gfCNCPoint3[12067] = {X 589.3965, Y 44.0652, Z -3.8333, A 0.000, B 0.000, C 0.000 }
gfCNCPoint3[12068] = {X 589.5012, Y 43.1533, Z -3.8333, A 0.000, B 0.000, C 0.000 }
gfCNCPoint3[12069] = {X 589.8014, Y 42.2858, Z -3.8333, A 0.000, B 0.000, C 0.000 }
gfCNCPoint3[12070] = {X 590.2828, Y 41.5042, Z -3.8333, A 0.000, B 0.000, C 0.000 }
gfCNCPoint3[12071] = {X 590.9225, Y 40.8459, Z -3.8333, A 0.000, B 0.000, C 0.000 }
gfCNCPoint3[12072] = {X 590.9230, Y 32.7095, Z -3.8333, A 0.000, B 0.000, C 0.000 }
gfCNCPoint3[12073] = {X 585.2975, Y 46.5912, Z -3.8333, A 0.000, B 0.000, C 0.000 }
gfCNCPoint3[12074] = {X 584.9414, Y 47.2678, Z -3.8333, A 0.000, B 0.000, C 0.000 }
gfCNCPoint3[12075] = {X 584.4675, Y 47.8677, Z -3.8333, A 0.000, B 0.000, C 0.000 }
gfCNCPoint3[12076] = {X 583.8918, Y 48.3708, Z -3.8333, A 0.000, B 0.000, C 0.000 }
gfCNCPoint3[12077] = {X 583.2338, Y 48.7600, Z -3.8333, A 0.000, B 0.000, C 0.000 }
gfCNCPoint3[12078] = {X 582.3250, Y 49.0678, Z -3.8333, A 0.000, B 0.000, C 0.000 }
gfCNCPoint3[12079] = {X 581.3699, Y 49.1592, Z -3.8333, A 0.000, B 0.000, C 0.000 }
gfCNCPoint3[12080] = {X 580.4192, Y 49.0293, Z -3.8333, A 0.000, B 0.000, C 0.000 }
gfCNCPoint3[12081] = {X 579.5236, Y 48.6850, Z -3.8333, A 0.000, B 0.000, C 0.000 }
gfCNCPoint3[12082] = {X 578.7306, Y 48.1448, Z -3.8333, A 0.000, B 0.000, C 0.000 }
gfCNCPoint3[12083] = {X 578.0826, Y 47.4372, Z -3.8333, A 0.000, B 0.000, C 0.000 }
gfCNCPoint3[12084] = {X 577.6138, Y 46.5999, Z -3.8333, A 0.000, B 0.000, C 0.000 }
gfCNCPoint3[12085] = {X 571.8585, Y 32.5267, Z -3.8333, A 0.000, B 0.000, C 0.000 }
gfCNCPoint3[12086] = {X 571.8589, Y 40.8461, Z -3.8333, A 0.000, B 0.000, C 0.000 }
gfCNCPoint3[12087] = {X 571.9195, Y 40.8953, Z -3.8333, A 0.000, B 0.000, C 0.000 }
gfCNCPoint3[12088] = {X 572.5327, Y 41.5413, Z -3.8333, A 0.000, B 0.000, C 0.000 }
gfCNCPoint3[12089] = {X 572.9944, Y 42.3029, Z -3.8333, A 0.000, B 0.000, C 0.000 }
gfCNCPoint3[12090] = {X 573.2833, Y 43.1454, Z -3.8333, A 0.000, B 0.000, C 0.000 }
gfCNCPoint3[12091] = {X 573.3863, Y 44.0301, Z -3.8333, A 0.000, B 0.000, C 0.000 }
gfCNCPoint3[12092] = {X 573.3864, Y 45.0000, Z -3.8333, A 0.000, B 0.000, C 0.000 }
gfCNCPoint3[12093] = {X 573.2821, Y 45.9257, Z -3.8333, A 0.000, B 0.000, C 0.000 }
gfCNCPoint3[12094] = {X 572.9745, Y 46.8050, Z -3.8333, A 0.000, B 0.000, C 0.000 }
gfCNCPoint3[12095] = {X 572.4788, Y 47.5937, Z -3.8333, A 0.000, B 0.000, C 0.000 }
gfCNCPoint3[12096] = {X 571.8201, Y 48.2524, Z -3.8333, A 0.000, B 0.000, C 0.000 }
gfCNCPoint3[12097] = {X 571.0314, Y 48.7480, Z -3.8333, A 0.000, B 0.000, C 0.000 }
gfCNCPoint3[12098] = {X 570.1521, Y 49.0557, Z -3.8333, A 0.000, B 0.000, C 0.000 }
gfCNCPoint3[12099] = {X 569.2264, Y 49.1600, Z -3.8333, A 0.000, B 0.000, C 0.000 }
gfCNCPoint3[12100] = {X 562.4443, Y 49.1600, Z -3.8333, A 0.000, B 0.000, C 0.000 }
gfCNCPoint3[12101] = {X 561.5186, Y 49.0557, Z -3.8333, A 0.000, B 0.000, C 0.000 }
gfCNCPoint3[12102] = {X 560.6393, Y 48.7480, Z -3.8333, A 0.000, B 0.000, C 0.000 }
gfCNCPoint3[12103] = {X 559.8506, Y 48.2524, Z -3.8333, A 0.000, B 0.000, C 0.000 }
gfCNCPoint3[12104] = {X 559.1919, Y 47.5937, Z -3.8333, A 0.000, B 0.000, C 0.000 }
gfCNCPoint3[12105] = {X 558.6963, Y 46.8050, Z -3.8333, A 0.000, B 0.000, C 0.000 }
gfCNCPoint3[12106] = {X 558.3886, Y 45.9257, Z -3.8333, A 0.000, B 0.000, C 0.000 }
gfCNCPoint3[12107] = {X 558.2843, Y 45.0000, Z -3.8333, A 0.000, B 0.000, C 0.000 }
gfCNCPoint3[12108] = {X 558.2843, Y 44.0653, Z -3.8333, A 0.000, B 0.000, C 0.000 }
gfCNCPoint3[12109] = {X 558.3888, Y 43.1529, Z -3.8333, A 0.000, B 0.000, C 0.000 }
gfCNCPoint3[12110] = {X 558.6893, Y 42.2852, Z -3.8333, A 0.000, B 0.000, C 0.000 }
gfCNCPoint3[12111] = {X 559.1714, Y 41.5036, Z -3.8333, A 0.000, B 0.000, C 0.000 }
gfCNCPoint3[12112] = {X 559.8121, Y 40.8457, Z -3.8333, A 0.000, B 0.000, C 0.000 }
gfCNCPoint3[12113] = {X 559.8121, Y 9.1554, Z -3.8333, A 0.000, B 0.000, C 0.000 }
gfCNCPoint3[12114] = {X 559.1745, Y 8.5058, Z -3.8333, A 0.000, B 0.000, C 0.000 }
gfCNCPoint3[12115] = {X 558.6934, Y 7.7331, Z -3.8333, A 0.000, B 0.000, C 0.000 }
gfCNCPoint3[12116] = {X 558.3919, Y 6.8743, Z -3.8333, A 0.000, B 0.000, C 0.000 }
gfCNCPoint3[12117] = {X 558.2845, Y 5.9704, Z -3.8333, A 0.000, B 0.000, C 0.000 }
gfCNCPoint3[12118] = {X 558.2843, Y 5.0000, Z -3.8333, A 0.000, B 0.000, C 0.000 }
gfCNCPoint3[12119] = {X 558.3886, Y 4.0743, Z -3.8333, A 0.000, B 0.000, C 0.000 }
gfCNCPoint3[12120] = {X 558.6963, Y 3.1950, Z -3.8333, A 0.000, B 0.000, C 0.000 }
gfCNCPoint3[12121] = {X 559.1919, Y 2.4063, Z -3.8333, A 0.000, B 0.000, C 0.000 }
gfCNCPoint3[12122] = {X 559.8506, Y 1.7476, Z -3.8333, A 0.000, B 0.000, C 0.000 }
gfCNCPoint3[12123] = {X 560.6393, Y 1.2520, Z -3.8333, A 0.000, B 0.000, C 0.000 }
gfCNCPoint3[12124] = {X 561.5186, Y 0.9443, Z -3.8333, A 0.000, B 0.000, C 0.000 }
gfCNCPoint3[12125] = {X 562.4443, Y 0.8400, Z -3.8333, A 0.000, B 0.000, C 0.000 }
gfCNCPoint3[12126] = {X 570.9376, Y 0.8400, Z -3.8333, A 0.000, B 0.000, C 0.000 }
gfCNCPoint3[12127] = {X 571.8632, Y 0.9443, Z -3.8333, A 0.000, B 0.000, C 0.000 }
gfCNCPoint3[12128] = {X 572.7425, Y 1.2520, Z -3.8333, A 0.000, B 0.000, C 0.000 }
gfCNCPoint3[12129] = {X 573.5313, Y 1.7476, Z -3.8333, A 0.000, B 0.000, C 0.000 }
gfCNCPoint3[12130] = {X 574.1900, Y 2.4063, Z -3.8333, A 0.000, B 0.000, C 0.000 }
gfCNCPoint3[12131] = {X 574.6856, Y 3.1950, Z -3.8333, A 0.000, B 0.000, C 0.000 }
gfCNCPoint3[12132] = {X 574.9933, Y 4.0743, Z -3.8333, A 0.000, B 0.000, C 0.000 }
gfCNCPoint3[12133] = {X 575.0976, Y 5.0000, Z -3.8333, A 0.000, B 0.000, C 0.000 }
gfCNCPoint3[12134] = {X 575.0976, Y 5.9342, Z -3.8333, A 0.000, B 0.000, C 0.000 }
gfCNCPoint3[12135] = {X 575.0212, Y 6.7277, Z -3.8333, A 0.000, B 0.000, C 0.000 }
gfCNCPoint3[12136] = {X 574.7948, Y 7.4920, Z -3.8333, A 0.000, B 0.000, C 0.000 }
gfCNCPoint3[12137] = {X 574.4268, Y 8.1991, Z -3.8333, A 0.000, B 0.000, C 0.000 }
gfCNCPoint3[12138] = {X 581.1907, Y 24.7935, Z -3.8333, A 0.000, B 0.000, C 0.000 }
gfCNCPoint3[12139] = {X 588.0240, Y 8.0814, Z -3.8333, A 0.000, B 0.000, C 0.000 }
gfCNCPoint3[12140] = {X 587.7001, Y 7.4166, Z -3.8333, A 0.000, B 0.000, C 0.000 }
gfCNCPoint3[12141] = {X 587.4990, Y 6.7051, Z -3.8333, A 0.000, B 0.000, C 0.000 }
gfCNCPoint3[12142] = {X 587.4271, Y 5.9692, Z -3.8333, A 0.000, B 0.000, C 0.000 }
gfCNCPoint3[12143] = {X 587.4270, Y 5.0000, Z -3.8333, A 0.000, B 0.000, C 0.000 }
gfCNCPoint3[12144] = {X 587.5313, Y 4.0743, Z -3.8333, A 0.000, B 0.000, C 0.000 }
gfCNCPoint3[12145] = {X 587.8389, Y 3.1950, Z -3.8333, A 0.000, B 0.000, C 0.000 }
gfCNCPoint3[12146] = {X 588.3345, Y 2.4063, Z -3.8333, A 0.000, B 0.000, C 0.000 }
gfCNCPoint3[12147] = {X 588.9932, Y 1.7476, Z -3.8333, A 0.000, B 0.000, C 0.000 }
gfCNCPoint3[12148] = {X 589.7820, Y 1.2520, Z -3.8333, A 0.000, B 0.000, C 0.000 }
gfCNCPoint3[12149] = {X 590.6613, Y 0.9443, Z -3.8333, A 0.000, B 0.000, C 0.000 }
gfCNCPoint3[12150] = {X 591.5870, Y 0.8400, Z -3.8333, A 0.000, B 0.000, C 0.000 }
gfCNCPoint3[12151] = {X 600.0000, Y 0.8400, Z -3.8333, A 0.000, B 0.000, C 0.000 }
gfCNCPoint3[12152] = {X 600.8244, Y 0.9225, Z -3.8333, A 0.000, B 0.000, C 0.000 }
gfCNCPoint3[12153] = {X 601.6162, Y 1.1668, Z -3.8333, A 0.000, B 0.000, C 0.000 }
gfCNCPoint3[12154] = {X 602.3438, Y 1.5631, Z -3.8333, A 0.000, B 0.000, C 0.000 }
gfCNCPoint3[12155] = {X 602.9784, Y 2.0958, Z -3.8333, A 0.000, B 0.000, C 0.000 }
gfCNCPoint3[12156] = {X 603.4949, Y 2.7436, Z -3.8333, A 0.000, B 0.000, C 0.000 }
gfCNCPoint3[12157] = {X 603.5999, Y 2.9153, Z -3.8333, A 0.000, B 0.000, C 0.000 }
gfCNCPoint3[12158] = {X 603.6965, Y 3.0918, Z -3.8333, A 0.000, B 0.000, C 0.000 }
gfCNCPoint3[12159] = {X 607.6965, Y 10.8407, Z -3.8333, A 0.000, B 0.000, C 0.000 }
gfCNCPoint3[12160] = {X 607.6965, Y 10.8407, Z -0.8333, A 0.000, B 0.000, C 0.000 }
gfCNCPoint3[12161] = {X 607.6965, Y 10.8407, Z 11.0000, A 0.000, B 0.000, C 0.000 }
gfCNCPoint3[12162] = {X 607.6965, Y 38.1642, Z 11.0000, A 0.000, B 0.000, C 0.000 }
gfCNCPoint3[12163] = {X 607.6965, Y 38.1642, Z -0.8333, A 0.000, B 0.000, C 0.000 }
gfCNCPoint3[12164] = {X 607.6965, Y 38.1642, Z -3.8333, A 0.000, B 0.000, C 0.000 }
gfCNCPoint3[12165] = {X 603.6965, Y 46.7268, Z -3.8333, A 0.000, B 0.000, C 0.000 }
gfCNCPoint3[12166] = {X 603.5704, Y 46.9745, Z -3.8333, A 0.000, B 0.000, C 0.000 }
gfCNCPoint3[12167] = {X 603.4277, Y 47.2130, Z -3.8333, A 0.000, B 0.000, C 0.000 }
gfCNCPoint3[12168] = {X 602.9211, Y 47.8484, Z -3.8333, A 0.000, B 0.000, C 0.000 }
gfCNCPoint3[12169] = {X 602.2987, Y 48.3708, Z -3.8333, A 0.000, B 0.000, C 0.000 }
gfCNCPoint3[12170] = {X 601.5851, Y 48.7595, Z -3.8333, A 0.000, B 0.000, C 0.000 }
gfCNCPoint3[12171] = {X 600.8086, Y 48.9991, Z -3.8333, A 0.000, B 0.000, C 0.000 }
gfCNCPoint3[12172] = {X 600.0000, Y 49.0800, Z -3.8333, A 0.000, B 0.000, C 0.000 }
gfCNCPoint3[12173] = {X 593.5565, Y 49.0800, Z -3.8333, A 0.000, B 0.000, C 0.000 }
gfCNCPoint3[12174] = {X 592.6486, Y 48.9777, Z -3.8333, A 0.000, B 0.000, C 0.000 }
gfCNCPoint3[12175] = {X 591.7863, Y 48.6760, Z -3.8333, A 0.000, B 0.000, C 0.000 }
gfCNCPoint3[12176] = {X 591.0127, Y 48.1899, Z -3.8333, A 0.000, B 0.000, C 0.000 }
gfCNCPoint3[12177] = {X 590.3667, Y 47.5438, Z -3.8333, A 0.000, B 0.000, C 0.000 }
gfCNCPoint3[12178] = {X 589.8806, Y 46.7702, Z -3.8333, A 0.000, B 0.000, C 0.000 }
gfCNCPoint3[12179] = {X 589.5788, Y 45.9079, Z -3.8333, A 0.000, B 0.000, C 0.000 }
gfCNCPoint3[12180] = {X 589.4765, Y 45.0000, Z -3.8333, A 0.000, B 0.000, C 0.000 }
gfCNCPoint3[12181] = {X 589.4765, Y 44.0656, Z -3.8333, A 0.000, B 0.000, C 0.000 }
gfCNCPoint3[12182] = {X 589.5734, Y 43.1967, Z -3.8333, A 0.000, B 0.000, C 0.000 }
gfCNCPoint3[12183] = {X 589.8514, Y 42.3678, Z -3.8333, A 0.000, B 0.000, C 0.000 }
gfCNCPoint3[12184] = {X 590.2980, Y 41.6162, Z -3.8333, A 0.000, B 0.000, C 0.000 }
gfCNCPoint3[12185] = {X 590.8930, Y 40.9757, Z -3.8333, A 0.000, B 0.000, C 0.000 }
gfCNCPoint3[12186] = {X 590.9473, Y 40.9293, Z -3.8333, A 0.000, B 0.000, C 0.000 }
gfCNCPoint3[12187] = {X 591.0025, Y 40.8838, Z -3.8333, A 0.000, B 0.000, C 0.000 }
gfCNCPoint3[12188] = {X 591.0030, Y 32.2990, Z -3.8333, A 0.000, B 0.000, C 0.000 }
gfCNCPoint3[12189] = {X 585.2236, Y 46.5606, Z -3.8333, A 0.000, B 0.000, C 0.000 }
gfCNCPoint3[12190] = {X 584.8743, Y 47.2242, Z -3.8333, A 0.000, B 0.000, C 0.000 }
gfCNCPoint3[12191] = {X 584.4095, Y 47.8125, Z -3.8333, A 0.000, B 0.000, C 0.000 }
gfCNCPoint3[12192] = {X 583.8449, Y 48.3059, Z -3.8333, A 0.000, B 0.000, C 0.000 }
gfCNCPoint3[12193] = {X 583.1996, Y 48.6877, Z -3.8333, A 0.000, B 0.000, C 0.000 }
gfCNCPoint3[12194] = {X 582.3082, Y 48.9895, Z -3.8333, A 0.000, B 0.000, C 0.000 }
gfCNCPoint3[12195] = {X 581.3715, Y 49.0792, Z -3.8333, A 0.000, B 0.000, C 0.000 }
gfCNCPoint3[12196] = {X 580.4391, Y 48.9518, Z -3.8333, A 0.000, B 0.000, C 0.000 }
gfCNCPoint3[12197] = {X 579.5607, Y 48.6142, Z -3.8333, A 0.000, B 0.000, C 0.000 }
gfCNCPoint3[12198] = {X 578.7830, Y 48.0843, Z -3.8333, A 0.000, B 0.000, C 0.000 }
gfCNCPoint3[12199] = {X 578.1474, Y 47.3903, Z -3.8333, A 0.000, B 0.000, C 0.000 }
gfCNCPoint3[12200] = {X 577.6877, Y 46.5692, Z -3.8333, A 0.000, B 0.000, C 0.000 }
gfCNCPoint3[12201] = {X 571.7785, Y 32.1197, Z -3.8333, A 0.000, B 0.000, C 0.000 }
gfCNCPoint3[12202] = {X 571.7789, Y 40.8842, Z -3.8333, A 0.000, B 0.000, C 0.000 }
gfCNCPoint3[12203] = {X 571.8684, Y 40.9569, Z -3.8333, A 0.000, B 0.000, C 0.000 }
gfCNCPoint3[12204] = {X 572.4695, Y 41.5903, Z -3.8333, A 0.000, B 0.000, C 0.000 }
gfCNCPoint3[12205] = {X 572.9221, Y 42.3372, Z -3.8333, A 0.000, B 0.000, C 0.000 }
gfCNCPoint3[12206] = {X 573.2053, Y 43.1633, Z -3.8333, A 0.000, B 0.000, C 0.000 }
gfCNCPoint3[12207] = {X 573.3063, Y 44.0308, Z -3.8333, A 0.000, B 0.000, C 0.000 }
gfCNCPoint3[12208] = {X 573.3064, Y 45.0000, Z -3.8333, A 0.000, B 0.000, C 0.000 }
gfCNCPoint3[12209] = {X 573.2041, Y 45.9079, Z -3.8333, A 0.000, B 0.000, C 0.000 }
gfCNCPoint3[12210] = {X 572.9024, Y 46.7702, Z -3.8333, A 0.000, B 0.000, C 0.000 }
gfCNCPoint3[12211] = {X 572.4163, Y 47.5438, Z -3.8333, A 0.000, B 0.000, C 0.000 }
gfCNCPoint3[12212] = {X 571.7703, Y 48.1899, Z -3.8333, A 0.000, B 0.000, C 0.000 }
gfCNCPoint3[12213] = {X 570.9967, Y 48.6760, Z -3.8333, A 0.000, B 0.000, C 0.000 }
gfCNCPoint3[12214] = {X 570.1343, Y 48.9777, Z -3.8333, A 0.000, B 0.000, C 0.000 }
gfCNCPoint3[12215] = {X 569.2264, Y 49.0800, Z -3.8333, A 0.000, B 0.000, C 0.000 }
gfCNCPoint3[12216] = {X 562.4443, Y 49.0800, Z -3.8333, A 0.000, B 0.000, C 0.000 }
gfCNCPoint3[12217] = {X 561.5364, Y 48.9777, Z -3.8333, A 0.000, B 0.000, C 0.000 }
gfCNCPoint3[12218] = {X 560.6741, Y 48.6760, Z -3.8333, A 0.000, B 0.000, C 0.000 }
gfCNCPoint3[12219] = {X 559.9005, Y 48.1899, Z -3.8333, A 0.000, B 0.000, C 0.000 }
gfCNCPoint3[12220] = {X 559.2544, Y 47.5438, Z -3.8333, A 0.000, B 0.000, C 0.000 }
gfCNCPoint3[12221] = {X 558.7683, Y 46.7702, Z -3.8333, A 0.000, B 0.000, C 0.000 }
gfCNCPoint3[12222] = {X 558.4666, Y 45.9079, Z -3.8333, A 0.000, B 0.000, C 0.000 }
gfCNCPoint3[12223] = {X 558.3643, Y 45.0000, Z -3.8333, A 0.000, B 0.000, C 0.000 }
gfCNCPoint3[12224] = {X 558.3643, Y 44.0656, Z -3.8333, A 0.000, B 0.000, C 0.000 }
gfCNCPoint3[12225] = {X 558.4689, Y 43.1615, Z -3.8333, A 0.000, B 0.000, C 0.000 }
gfCNCPoint3[12226] = {X 558.7697, Y 42.3025, Z -3.8333, A 0.000, B 0.000, C 0.000 }
gfCNCPoint3[12227] = {X 559.2519, Y 41.5306, Z -3.8333, A 0.000, B 0.000, C 0.000 }
gfCNCPoint3[12228] = {X 559.8921, Y 40.8836, Z -3.8333, A 0.000, B 0.000, C 0.000 }
gfCNCPoint3[12229] = {X 559.8921, Y 9.1172, Z -3.8333, A 0.000, B 0.000, C 0.000 }
gfCNCPoint3[12230] = {X 559.2550, Y 8.4786, Z -3.8333, A 0.000, B 0.000, C 0.000 }
gfCNCPoint3[12231] = {X 558.7738, Y 7.7155, Z -3.8333, A 0.000, B 0.000, C 0.000 }
gfCNCPoint3[12232] = {X 558.4720, Y 6.8654, Z -3.8333, A 0.000, B 0.000, C 0.000 }
gfCNCPoint3[12233] = {X 558.3645, Y 5.9697, Z -3.8333, A 0.000, B 0.000, C 0.000 }
gfCNCPoint3[12234] = {X 558.3643, Y 5.0000, Z -3.8333, A 0.000, B 0.000, C 0.000 }
gfCNCPoint3[12235] = {X 558.4666, Y 4.0921, Z -3.8333, A 0.000, B 0.000, C 0.000 }
gfCNCPoint3[12236] = {X 558.7683, Y 3.2298, Z -3.8333, A 0.000, B 0.000, C 0.000 }
gfCNCPoint3[12237] = {X 559.2544, Y 2.4562, Z -3.8333, A 0.000, B 0.000, C 0.000 }
gfCNCPoint3[12238] = {X 559.9005, Y 1.8101, Z -3.8333, A 0.000, B 0.000, C 0.000 }
gfCNCPoint3[12239] = {X 560.6741, Y 1.3240, Z -3.8333, A 0.000, B 0.000, C 0.000 }
gfCNCPoint3[12240] = {X 561.5364, Y 1.0223, Z -3.8333, A 0.000, B 0.000, C 0.000 }
gfCNCPoint3[12241] = {X 562.4443, Y 0.9200, Z -3.8333, A 0.000, B 0.000, C 0.000 }
gfCNCPoint3[12242] = {X 570.9376, Y 0.9200, Z -3.8333, A 0.000, B 0.000, C 0.000 }
gfCNCPoint3[12243] = {X 571.8454, Y 1.0223, Z -3.8333, A 0.000, B 0.000, C 0.000 }
gfCNCPoint3[12244] = {X 572.7078, Y 1.3240, Z -3.8333, A 0.000, B 0.000, C 0.000 }
gfCNCPoint3[12245] = {X 573.4814, Y 1.8101, Z -3.8333, A 0.000, B 0.000, C 0.000 }
gfCNCPoint3[12246] = {X 574.1274, Y 2.4562, Z -3.8333, A 0.000, B 0.000, C 0.000 }
gfCNCPoint3[12247] = {X 574.6135, Y 3.2298, Z -3.8333, A 0.000, B 0.000, C 0.000 }
gfCNCPoint3[12248] = {X 574.9153, Y 4.0921, Z -3.8333, A 0.000, B 0.000, C 0.000 }
gfCNCPoint3[12249] = {X 575.0176, Y 5.0000, Z -3.8333, A 0.000, B 0.000, C 0.000 }
gfCNCPoint3[12250] = {X 575.0176, Y 5.9342, Z -3.8333, A 0.000, B 0.000, C 0.000 }
gfCNCPoint3[12251] = {X 574.9500, Y 6.6737, Z -3.8333, A 0.000, B 0.000, C 0.000 }
gfCNCPoint3[12252] = {X 574.7495, Y 7.3887, Z -3.8333, A 0.000, B 0.000, C 0.000 }
gfCNCPoint3[12253] = {X 574.4227, Y 8.0554, Z -3.8333, A 0.000, B 0.000, C 0.000 }
gfCNCPoint3[12254] = {X 574.3783, Y 8.1266, Z -3.8333, A 0.000, B 0.000, C 0.000 }
gfCNCPoint3[12255] = {X 574.3325, Y 8.1969, Z -3.8333, A 0.000, B 0.000, C 0.000 }
gfCNCPoint3[12256] = {X 574.3580, Y 8.2413, Z -3.8333, A 0.000, B 0.000, C 0.000 }
gfCNCPoint3[12257] = {X 581.1906, Y 25.0052, Z -3.8333, A 0.000, B 0.000, C 0.000 }
gfCNCPoint3[12258] = {X 588.1133, Y 8.0742, Z -3.8333, A 0.000, B 0.000, C 0.000 }
gfCNCPoint3[12259] = {X 588.0738, Y 8.0088, Z -3.8333, A 0.000, B 0.000, C 0.000 }
gfCNCPoint3[12260] = {X 588.0356, Y 7.9426, Z -3.8333, A 0.000, B 0.000, C 0.000 }
gfCNCPoint3[12261] = {X 587.7487, Y 7.3176, Z -3.8333, A 0.000, B 0.000, C 0.000 }
gfCNCPoint3[12262] = {X 587.5708, Y 6.6532, Z -3.8333, A 0.000, B 0.000, C 0.000 }
gfCNCPoint3[12263] = {X 587.5071, Y 5.9685, Z -3.8333, A 0.000, B 0.000, C 0.000 }
gfCNCPoint3[12264] = {X 587.5070, Y 5.0000, Z -3.8333, A 0.000, B 0.000, C 0.000 }
gfCNCPoint3[12265] = {X 587.6092, Y 4.0921, Z -3.8333, A 0.000, B 0.000, C 0.000 }
gfCNCPoint3[12266] = {X 587.9110, Y 3.2298, Z -3.8333, A 0.000, B 0.000, C 0.000 }
gfCNCPoint3[12267] = {X 588.3971, Y 2.4562, Z -3.8333, A 0.000, B 0.000, C 0.000 }
gfCNCPoint3[12268] = {X 589.0431, Y 1.8101, Z -3.8333, A 0.000, B 0.000, C 0.000 }
gfCNCPoint3[12269] = {X 589.8167, Y 1.3240, Z -3.8333, A 0.000, B 0.000, C 0.000 }
gfCNCPoint3[12270] = {X 590.6791, Y 1.0223, Z -3.8333, A 0.000, B 0.000, C 0.000 }
gfCNCPoint3[12271] = {X 591.5870, Y 0.9200, Z -3.8333, A 0.000, B 0.000, C 0.000 }
gfCNCPoint3[12272] = {X 600.0000, Y 0.9200, Z -3.8333, A 0.000, B 0.000, C 0.000 }
gfCNCPoint3[12273] = {X 600.8086, Y 1.0009, Z -3.8333, A 0.000, B 0.000, C 0.000 }
gfCNCPoint3[12274] = {X 601.5851, Y 1.2405, Z -3.8333, A 0.000, B 0.000, C 0.000 }
gfCNCPoint3[12275] = {X 602.2987, Y 1.6292, Z -3.8333, A 0.000, B 0.000, C 0.000 }
gfCNCPoint3[12276] = {X 602.9211, Y 2.1516, Z -3.8333, A 0.000, B 0.000, C 0.000 }
gfCNCPoint3[12277] = {X 603.4277, Y 2.7870, Z -3.8333, A 0.000, B 0.000, C 0.000 }
gfCNCPoint3[12278] = {X 603.5704, Y 3.0255, Z -3.8333, A 0.000, B 0.000, C 0.000 }
gfCNCPoint3[12279] = {X 603.6965, Y 3.2732, Z -3.8333, A 0.000, B 0.000, C 0.000 }
gfCNCPoint3[12280] = {X 607.6965, Y 11.8358, Z -3.8333, A 0.000, B 0.000, C 0.000 }
gfCNCPoint3[12281] = {X 607.6965, Y 11.8358, Z -0.8333, A 0.000, B 0.000, C 0.000 }
gfCNCPoint3[12282] = {X 607.6965, Y 11.8358, Z 11.0000, A 0.000, B 0.000, C 0.000 }
gfCNCPoint3[12283] = {X 607.6965, Y 36.8530, Z 11.0000, A 0.000, B 0.000, C 0.000 }
gfCNCPoint3[12284] = {X 607.6965, Y 36.8530, Z -0.8333, A 0.000, B 0.000, C 0.000 }
gfCNCPoint3[12285] = {X 607.6965, Y 36.8530, Z -3.8333, A 0.000, B 0.000, C 0.000 }
gfCNCPoint3[12286] = {X 603.6965, Y 46.5283, Z -3.8333, A 0.000, B 0.000, C 0.000 }
gfCNCPoint3[12287] = {X 603.5431, Y 46.8565, Z -3.8333, A 0.000, B 0.000, C 0.000 }
gfCNCPoint3[12288] = {X 603.3605, Y 47.1696, Z -3.8333, A 0.000, B 0.000, C 0.000 }
gfCNCPoint3[12289] = {X 602.8639, Y 47.7925, Z -3.8333, A 0.000, B 0.000, C 0.000 }
gfCNCPoint3[12290] = {X 602.2536, Y 48.3047, Z -3.8333, A 0.000, B 0.000, C 0.000 }
gfCNCPoint3[12291] = {X 601.5540, Y 48.6858, Z -3.8333, A 0.000, B 0.000, C 0.000 }
gfCNCPoint3[12292] = {X 600.7927, Y 48.9207, Z -3.8333, A 0.000, B 0.000, C 0.000 }
gfCNCPoint3[12293] = {X 600.0000, Y 49.0000, Z -3.8333, A 0.000, B 0.000, C 0.000 }
gfCNCPoint3[12294] = {X 593.5565, Y 49.0000, Z -3.8333, A 0.000, B 0.000, C 0.000 }
gfCNCPoint3[12295] = {X 592.6664, Y 48.8997, Z -3.8333, A 0.000, B 0.000, C 0.000 }
gfCNCPoint3[12296] = {X 591.8210, Y 48.6039, Z -3.8333, A 0.000, B 0.000, C 0.000 }
gfCNCPoint3[12297] = {X 591.0626, Y 48.1273, Z -3.8333, A 0.000, B 0.000, C 0.000 }
gfCNCPoint3[12298] = {X 590.4292, Y 47.4940, Z -3.8333, A 0.000, B 0.000, C 0.000 }
gfCNCPoint3[12299] = {X 589.9527, Y 46.7355, Z -3.8333, A 0.000, B 0.000, C 0.000 }
gfCNCPoint3[12300] = {X 589.6568, Y 45.8901, Z -3.8333, A 0.000, B 0.000, C 0.000 }
gfCNCPoint3[12301] = {X 589.5565, Y 45.0000, Z -3.8333, A 0.000, B 0.000, C 0.000 }
gfCNCPoint3[12302] = {X 589.5565, Y 44.0660, Z -3.8333, A 0.000, B 0.000, C 0.000 }
gfCNCPoint3[12303] = {X 589.6515, Y 43.2140, Z -3.8333, A 0.000, B 0.000, C 0.000 }
gfCNCPoint3[12304] = {X 589.9241, Y 42.4012, Z -3.8333, A 0.000, B 0.000, C 0.000 }
gfCNCPoint3[12305] = {X 590.3620, Y 41.6642, Z -3.8333, A 0.000, B 0.000, C 0.000 }
gfCNCPoint3[12306] = {X 590.9455, Y 41.0361, Z -3.8333, A 0.000, B 0.000, C 0.000 }
gfCNCPoint3[12307] = {X 591.0133, Y 40.9784, Z -3.8333, A 0.000, B 0.000, C 0.000 }
gfCNCPoint3[12308] = {X 591.0824, Y 40.9222, Z -3.8333, A 0.000, B 0.000, C 0.000 }
gfCNCPoint3[12309] = {X 591.0844, Y 40.3075, Z -3.8333, A 0.000, B 0.000, C 0.000 }
gfCNCPoint3[12310] = {X 591.0830, Y 32.0431, Z -3.8333, A 0.000, B 0.000, C 0.000 }
gfCNCPoint3[12311] = {X 590.9675, Y 32.1736, Z -3.8333, A 0.000, B 0.000, C 0.000 }
gfCNCPoint3[12312] = {X 590.3126, Y 33.7898, Z -3.8333, A 0.000, B 0.000, C 0.000 }
gfCNCPoint3[12313] = {X 585.1497, Y 46.5300, Z -3.8333, A 0.000, B 0.000, C 0.000 }
gfCNCPoint3[12314] = {X 584.8073, Y 47.1805, Z -3.8333, A 0.000, B 0.000, C 0.000 }
gfCNCPoint3[12315] = {X 584.3516, Y 47.7574, Z -3.8333, A 0.000, B 0.000, C 0.000 }
gfCNCPoint3[12316] = {X 583.7980, Y 48.2411, Z -3.8333, A 0.000, B 0.000, C 0.000 }
gfCNCPoint3[12317] = {X 583.1653, Y 48.6154, Z -3.8333, A 0.000, B 0.000, C 0.000 }
gfCNCPoint3[12318] = {X 582.2878, Y 48.9121, Z -3.8333, A 0.000, B 0.000, C 0.000 }
gfCNCPoint3[12319] = {X 581.3656, Y 48.9990, Z -3.8333, A 0.000, B 0.000, C 0.000 }
gfCNCPoint3[12320] = {X 580.4480, Y 48.8715, Z -3.8333, A 0.000, B 0.000, C 0.000 }
gfCNCPoint3[12321] = {X 579.5845, Y 48.5363, Z -3.8333, A 0.000, B 0.000, C 0.000 }
gfCNCPoint3[12322] = {X 578.8212, Y 48.0115, Z -3.8333, A 0.000, B 0.000, C 0.000 }
gfCNCPoint3[12323] = {X 578.1990, Y 47.3251, Z -3.8333, A 0.000, B 0.000, C 0.000 }
gfCNCPoint3[12324] = {X 577.7515, Y 46.5141, Z -3.8333, A 0.000, B 0.000, C 0.000 }
gfCNCPoint3[12325] = {X 571.6985, Y 31.7127, Z -3.8333, A 0.000, B 0.000, C 0.000 }
gfCNCPoint3[12326] = {X 571.6989, Y 40.9223, Z -3.8333, A 0.000, B 0.000, C 0.000 }
gfCNCPoint3[12327] = {X 571.8378, Y 41.0359, Z -3.8333, A 0.000, B 0.000, C 0.000 }
gfCNCPoint3[12328] = {X 572.4238, Y 41.6624, Z -3.8333, A 0.000, B 0.000, C 0.000 }
gfCNCPoint3[12329] = {X 572.8627, Y 42.3994, Z -3.8333, A 0.000, B 0.000, C 0.000 }
gfCNCPoint3[12330] = {X 573.1345, Y 43.2131, Z -3.8333, A 0.000, B 0.000, C 0.000 }
gfCNCPoint3[12331] = {X 573.2264, Y 44.0660, Z -3.8333, A 0.000, B 0.000, C 0.000 }
gfCNCPoint3[12332] = {X 573.2264, Y 45.0000, Z -3.8333, A 0.000, B 0.000, C 0.000 }
gfCNCPoint3[12333] = {X 573.1261, Y 45.8901, Z -3.8333, A 0.000, B 0.000, C 0.000 }
gfCNCPoint3[12334] = {X 572.8303, Y 46.7355, Z -3.8333, A 0.000, B 0.000, C 0.000 }
gfCNCPoint3[12335] = {X 572.3538, Y 47.4940, Z -3.8333, A 0.000, B 0.000, C 0.000 }
gfCNCPoint3[12336] = {X 571.7204, Y 48.1273, Z -3.8333, A 0.000, B 0.000, C 0.000 }
gfCNCPoint3[12337] = {X 570.9620, Y 48.6039, Z -3.8333, A 0.000, B 0.000, C 0.000 }
gfCNCPoint3[12338] = {X 570.1165, Y 48.8997, Z -3.8333, A 0.000, B 0.000, C 0.000 }
gfCNCPoint3[12339] = {X 569.2264, Y 49.0000, Z -3.8333, A 0.000, B 0.000, C 0.000 }
gfCNCPoint3[12340] = {X 562.4443, Y 49.0000, Z -3.8333, A 0.000, B 0.000, C 0.000 }
gfCNCPoint3[12341] = {X 561.5542, Y 48.8997, Z -3.8333, A 0.000, B 0.000, C 0.000 }
gfCNCPoint3[12342] = {X 560.7088, Y 48.6039, Z -3.8333, A 0.000, B 0.000, C 0.000 }
gfCNCPoint3[12343] = {X 559.9503, Y 48.1273, Z -3.8333, A 0.000, B 0.000, C 0.000 }
gfCNCPoint3[12344] = {X 559.3170, Y 47.4940, Z -3.8333, A 0.000, B 0.000, C 0.000 }
gfCNCPoint3[12345] = {X 558.8404, Y 46.7355, Z -3.8333, A 0.000, B 0.000, C 0.000 }
gfCNCPoint3[12346] = {X 558.5446, Y 45.8901, Z -3.8333, A 0.000, B 0.000, C 0.000 }
gfCNCPoint3[12347] = {X 558.4443, Y 45.0000, Z -3.8333, A 0.000, B 0.000, C 0.000 }
gfCNCPoint3[12348] = {X 558.4443, Y 44.0660, Z -3.8333, A 0.000, B 0.000, C 0.000 }
gfCNCPoint3[12349] = {X 558.5490, Y 43.1702, Z -3.8333, A 0.000, B 0.000, C 0.000 }
gfCNCPoint3[12350] = {X 558.8501, Y 42.3200, Z -3.8333, A 0.000, B 0.000, C 0.000 }
gfCNCPoint3[12351] = {X 559.3325, Y 41.5579, Z -3.8333, A 0.000, B 0.000, C 0.000 }
gfCNCPoint3[12352] = {X 559.9721, Y 40.9221, Z -3.8333, A 0.000, B 0.000, C 0.000 }
gfCNCPoint3[12353] = {X 559.9721, Y 9.0786, Z -3.8333, A 0.000, B 0.000, C 0.000 }
gfCNCPoint3[12354] = {X 559.3300, Y 8.4442, Z -3.8333, A 0.000, B 0.000, C 0.000 }
gfCNCPoint3[12355] = {X 558.8464, Y 7.6820, Z -3.8333, A 0.000, B 0.000, C 0.000 }
gfCNCPoint3[12356] = {X 558.5461, Y 6.8308, Z -3.8333, A 0.000, B 0.000, C 0.000 }
gfCNCPoint3[12357] = {X 558.4443, Y 5.9339, Z -3.8333, A 0.000, B 0.000, C 0.000 }
gfCNCPoint3[12358] = {X 558.4443, Y 5.0000, Z -3.8333, A 0.000, B 0.000, C 0.000 }
gfCNCPoint3[12359] = {X 558.5446, Y 4.1099, Z -3.8333, A 0.000, B 0.000, C 0.000 }
gfCNCPoint3[12360] = {X 558.8404, Y 3.2645, Z -3.8333, A 0.000, B 0.000, C 0.000 }
gfCNCPoint3[12361] = {X 559.3170, Y 2.5060, Z -3.8333, A 0.000, B 0.000, C 0.000 }
gfCNCPoint3[12362] = {X 559.9503, Y 1.8727, Z -3.8333, A 0.000, B 0.000, C 0.000 }
gfCNCPoint3[12363] = {X 560.7088, Y 1.3961, Z -3.8333, A 0.000, B 0.000, C 0.000 }
gfCNCPoint3[12364] = {X 561.5542, Y 1.1003, Z -3.8333, A 0.000, B 0.000, C 0.000 }
gfCNCPoint3[12365] = {X 562.4443, Y 1.0000, Z -3.8333, A 0.000, B 0.000, C 0.000 }
gfCNCPoint3[12366] = {X 570.9376, Y 1.0000, Z -3.8333, A 0.000, B 0.000, C 0.000 }
gfCNCPoint3[12367] = {X 571.8276, Y 1.1003, Z -3.8333, A 0.000, B 0.000, C 0.000 }
gfCNCPoint3[12368] = {X 572.6731, Y 1.3961, Z -3.8333, A 0.000, B 0.000, C 0.000 }
gfCNCPoint3[12369] = {X 573.4315, Y 1.8727, Z -3.8333, A 0.000, B 0.000, C 0.000 }
gfCNCPoint3[12370] = {X 574.0649, Y 2.5060, Z -3.8333, A 0.000, B 0.000, C 0.000 }
gfCNCPoint3[12371] = {X 574.5414, Y 3.2645, Z -3.8333, A 0.000, B 0.000, C 0.000 }
gfCNCPoint3[12372] = {X 574.8373, Y 4.1099, Z -3.8333, A 0.000, B 0.000, C 0.000 }
gfCNCPoint3[12373] = {X 574.9376, Y 5.0000, Z -3.8333, A 0.000, B 0.000, C 0.000 }
gfCNCPoint3[12374] = {X 574.9372, Y 5.9858, Z -3.8333, A 0.000, B 0.000, C 0.000 }
gfCNCPoint3[12375] = {X 574.8649, Y 6.6930, Z -3.8333, A 0.000, B 0.000, C 0.000 }
gfCNCPoint3[12376] = {X 574.6685, Y 7.3762, Z -3.8333, A 0.000, B 0.000, C 0.000 }
gfCNCPoint3[12377] = {X 574.3544, Y 8.0138, Z -3.8333, A 0.000, B 0.000, C 0.000 }
gfCNCPoint3[12378] = {X 574.2918, Y 8.1133, Z -3.8333, A 0.000, B 0.000, C 0.000 }
gfCNCPoint3[12379] = {X 574.2264, Y 8.2108, Z -3.8333, A 0.000, B 0.000, C 0.000 }
gfCNCPoint3[12380] = {X 574.2609, Y 8.2359, Z -3.8333, A 0.000, B 0.000, C 0.000 }
gfCNCPoint3[12381] = {X 574.2841, Y 8.2718, Z -3.8333, A 0.000, B 0.000, C 0.000 }
gfCNCPoint3[12382] = {X 574.9161, Y 9.8081, Z -3.8333, A 0.000, B 0.000, C 0.000 }
gfCNCPoint3[12383] = {X 581.1904, Y 25.2169, Z -3.8333, A 0.000, B 0.000, C 0.000 }
gfCNCPoint3[12384] = {X 588.2029, Y 8.0666, Z -3.8333, A 0.000, B 0.000, C 0.000 }
gfCNCPoint3[12385] = {X 588.1531, Y 7.9855, Z -3.8333, A 0.000, B 0.000, C 0.000 }
gfCNCPoint3[12386] = {X 588.1052, Y 7.9032, Z -3.8333, A 0.000, B 0.000, C 0.000 }
gfCNCPoint3[12387] = {X 587.8201, Y 7.2798, Z -3.8333, A 0.000, B 0.000, C 0.000 }
gfCNCPoint3[12388] = {X 587.6457, Y 6.6169, Z -3.8333, A 0.000, B 0.000, C 0.000 }
gfCNCPoint3[12389] = {X 587.5870, Y 5.9340, Z -3.8333, A 0.000, B 0.000, C 0.000 }
gfCNCPoint3[12390] = {X 587.5870, Y 5.0000, Z -3.8333, A 0.000, B 0.000, C 0.000 }
gfCNCPoint3[12391] = {X 587.6872, Y 4.1099, Z -3.8333, A 0.000, B 0.000, C 0.000 }
gfCNCPoint3[12392] = {X 587.9831, Y 3.2645, Z -3.8333, A 0.000, B 0.000, C 0.000 }
gfCNCPoint3[12393] = {X 588.4596, Y 2.5060, Z -3.8333, A 0.000, B 0.000, C 0.000 }
gfCNCPoint3[12394] = {X 589.0930, Y 1.8727, Z -3.8333, A 0.000, B 0.000, C 0.000 }
gfCNCPoint3[12395] = {X 589.8514, Y 1.3961, Z -3.8333, A 0.000, B 0.000, C 0.000 }
gfCNCPoint3[12396] = {X 590.6969, Y 1.1003, Z -3.8333, A 0.000, B 0.000, C 0.000 }
gfCNCPoint3[12397] = {X 591.5870, Y 1.0000, Z -3.8333, A 0.000, B 0.000, C 0.000 }
gfCNCPoint3[12398] = {X 600.0000, Y 1.0000, Z -3.8333, A 0.000, B 0.000, C 0.000 }
gfCNCPoint3[12399] = {X 600.7927, Y 1.0793, Z -3.8333, A 0.000, B 0.000, C 0.000 }
gfCNCPoint3[12400] = {X 601.5540, Y 1.3142, Z -3.8333, A 0.000, B 0.000, C 0.000 }
gfCNCPoint3[12401] = {X 602.2536, Y 1.6953, Z -3.8333, A 0.000, B 0.000, C 0.000 }
gfCNCPoint3[12402] = {X 602.8639, Y 2.2075, Z -3.8333, A 0.000, B 0.000, C 0.000 }
gfCNCPoint3[12403] = {X 603.3605, Y 2.8304, Z -3.8333, A 0.000, B 0.000, C 0.000 }
gfCNCPoint3[12404] = {X 603.5431, Y 3.1435, Z -3.8333, A 0.000, B 0.000, C 0.000 }
gfCNCPoint3[12405] = {X 603.6965, Y 3.4717, Z -3.8333, A 0.000, B 0.000, C 0.000 }
gfCNCPoint3[12406] = {X 607.6965, Y 13.1470, Z -3.8333, A 0.000, B 0.000, C 0.000 }
gfCNCPoint3[12407] = {X 607.6965, Y 13.1470, Z -0.8333, A 0.000, B 0.000, C 0.000 }
gfCNCPoint3[12408] = {X 607.6965, Y 13.1470, Z 11.0000, A 0.000, B 0.000, C 0.000 }
gfCNCPoint3[12409] = {X 448.7130, Y 19.7816, Z 11.0000, A 0.000, B 0.000, C 0.000 }
gfCNCPoint3[12410] = {X 448.7130, Y 19.7816, Z 0.0000, A 0.000, B 0.000, C 0.000 }
gfCNCPoint3[12411] = {X 444.0413, Y 19.7814, Z -1.2518, A 0.000, B 0.000, C 0.000 }
gfCNCPoint3[12412] = {X 443.3488, Y 19.7976, Z -1.4374, A 0.000, B 0.000, C 0.000 }
gfCNCPoint3[12413] = {X 442.7485, Y 19.8046, Z -1.5982, A 0.000, B 0.000, C 0.000 }
gfCNCPoint3[12414] = {X 442.0368, Y 19.9278, Z -1.7918, A 0.000, B 0.000, C 0.000 }
gfCNCPoint3[12415] = {X 441.4692, Y 20.1231, Z -1.9526, A 0.000, B 0.000, C 0.000 }
gfCNCPoint3[12416] = {X 441.3663, Y 20.1584, Z -1.9818, A 0.000, B 0.000, C 0.000 }
gfCNCPoint3[12417] = {X 441.3334, Y 20.2621, Z -2.0109, A 0.000, B 0.000, C 0.000 }
gfCNCPoint3[12418] = {X 441.1885, Y 20.7177, Z -2.1390, A 0.000, B 0.000, C 0.000 }
gfCNCPoint3[12419] = {X 441.1547, Y 21.8885, Z -2.4528, A 0.000, B 0.000, C 0.000 }
gfCNCPoint3[12420] = {X 441.2731, Y 22.3517, Z -2.5810, A 0.000, B 0.000, C 0.000 }
gfCNCPoint3[12421] = {X 441.5022, Y 22.4267, Z -2.6455, A 0.000, B 0.000, C 0.000 }
gfCNCPoint3[12422] = {X 441.7422, Y 22.4486, Z -2.7101, A 0.000, B 0.000, C 0.000 }
gfCNCPoint3[12423] = {X 442.9926, Y 22.5628, Z -3.0465, A 0.000, B 0.000, C 0.000 }
gfCNCPoint3[12424] = {X 443.1348, Y 22.5685, Z -3.0847, A 0.000, B 0.000, C 0.000 }
gfCNCPoint3[12425] = {X 444.3942, Y 22.5560, Z -3.4222, A 0.000, B 0.000, C 0.000 }
gfCNCPoint3[12426] = {X 445.9287, Y 22.5560, Z -3.8333, A 0.000, B 0.000, C 0.000 }
gfCNCPoint3[12427] = {X 450.1184, Y 22.5560, Z -3.8333, A 0.000, B 0.000, C 0.000 }
gfCNCPoint3[12428] = {X 450.1184, Y 19.7817, Z -3.8333, A 0.000, B 0.000, C 0.000 }
gfCNCPoint3[12429] = {X 444.0413, Y 19.7814, Z -3.8333, A 0.000, B 0.000, C 0.000 }
gfCNCPoint3[12430] = {X 443.3488, Y 19.7976, Z -3.8333, A 0.000, B 0.000, C 0.000 }
gfCNCPoint3[12431] = {X 442.3959, Y 19.8851, Z -3.8333, A 0.000, B 0.000, C 0.000 }
gfCNCPoint3[12432] = {X 441.4692, Y 20.1231, Z -3.8333, A 0.000, B 0.000, C 0.000 }
gfCNCPoint3[12433] = {X 441.3848, Y 20.1765, Z -3.8333, A 0.000, B 0.000, C 0.000 }
gfCNCPoint3[12434] = {X 441.3334, Y 20.2621, Z -3.8333, A 0.000, B 0.000, C 0.000 }
gfCNCPoint3[12435] = {X 441.1831, Y 20.9508, Z -3.8333, A 0.000, B 0.000, C 0.000 }
gfCNCPoint3[12436] = {X 441.1628, Y 21.6555, Z -3.8333, A 0.000, B 0.000, C 0.000 }
gfCNCPoint3[12437] = {X 441.2731, Y 22.3517, Z -3.8333, A 0.000, B 0.000, C 0.000 }
gfCNCPoint3[12438] = {X 441.5049, Y 22.4134, Z -3.8333, A 0.000, B 0.000, C 0.000 }
gfCNCPoint3[12439] = {X 441.7422, Y 22.4486, Z -3.8333, A 0.000, B 0.000, C 0.000 }
gfCNCPoint3[12440] = {X 443.0669, Y 22.5359, Z -3.8333, A 0.000, B 0.000, C 0.000 }
gfCNCPoint3[12441] = {X 444.3942, Y 22.5560, Z -3.8333, A 0.000, B 0.000, C 0.000 }
gfCNCPoint3[12442] = {X 445.9287, Y 22.5560, Z -3.8333, A 0.000, B 0.000, C 0.000 }
gfCNCPoint3[12443] = {X 441.9439, Y 22.2874, Z -3.8333, A 0.000, B 0.000, C 0.000 }
gfCNCPoint3[12444] = {X 445.9287, Y 22.6360, Z -3.8333, A 0.000, B 0.000, C 0.000 }
gfCNCPoint3[12445] = {X 450.1984, Y 22.6360, Z -3.8333, A 0.000, B 0.000, C 0.000 }
gfCNCPoint3[12446] = {X 450.1984, Y 19.7017, Z -3.8333, A 0.000, B 0.000, C 0.000 }
gfCNCPoint3[12447] = {X 444.0404, Y 19.7014, Z -3.8333, A 0.000, B 0.000, C 0.000 }
gfCNCPoint3[12448] = {X 443.3498, Y 19.7176, Z -3.8333, A 0.000, B 0.000, C 0.000 }
gfCNCPoint3[12449] = {X 442.3832, Y 19.8061, Z -3.8333, A 0.000, B 0.000, C 0.000 }
gfCNCPoint3[12450] = {X 441.4431, Y 20.0474, Z -3.8333, A 0.000, B 0.000, C 0.000 }
gfCNCPoint3[12451] = {X 441.3275, Y 20.1206, Z -3.8333, A 0.000, B 0.000, C 0.000 }
gfCNCPoint3[12452] = {X 441.2571, Y 20.2378, Z -3.8333, A 0.000, B 0.000, C 0.000 }
gfCNCPoint3[12453] = {X 441.1019, Y 20.9555, Z -3.8333, A 0.000, B 0.000, C 0.000 }
gfCNCPoint3[12454] = {X 441.0849, Y 21.6896, Z -3.8333, A 0.000, B 0.000, C 0.000 }
gfCNCPoint3[12455] = {X 441.2066, Y 22.4137, Z -3.8333, A 0.000, B 0.000, C 0.000 }
gfCNCPoint3[12456] = {X 441.4673, Y 22.4872, Z -3.8333, A 0.000, B 0.000, C 0.000 }
gfCNCPoint3[12457] = {X 441.7350, Y 22.5283, Z -3.8333, A 0.000, B 0.000, C 0.000 }
gfCNCPoint3[12458] = {X 443.0624, Y 22.6157, Z -3.8333, A 0.000, B 0.000, C 0.000 }
gfCNCPoint3[12459] = {X 444.3927, Y 22.6360, Z -3.8333, A 0.000, B 0.000, C 0.000 }
gfCNCPoint3[12460] = {X 445.9287, Y 22.6360, Z -3.8333, A 0.000, B 0.000, C 0.000 }
gfCNCPoint3[12461] = {X 449.9135, Y 22.2874, Z -3.8333, A 0.000, B 0.000, C 0.000 }
gfCNCPoint3[12462] = {X 441.9439, Y 22.3674, Z -3.8333, A 0.000, B 0.000, C 0.000 }
gfCNCPoint3[12463] = {X 445.9287, Y 22.7160, Z -3.8333, A 0.000, B 0.000, C 0.000 }
gfCNCPoint3[12464] = {X 450.2784, Y 22.7160, Z -3.8333, A 0.000, B 0.000, C 0.000 }
gfCNCPoint3[12465] = {X 450.2784, Y 19.6217, Z -3.8333, A 0.000, B 0.000, C 0.000 }
gfCNCPoint3[12466] = {X 444.0395, Y 19.6214, Z -3.8333, A 0.000, B 0.000, C 0.000 }
gfCNCPoint3[12467] = {X 443.3484, Y 19.6376, Z -3.8333, A 0.000, B 0.000, C 0.000 }
gfCNCPoint3[12468] = {X 442.3693, Y 19.7273, Z -3.8333, A 0.000, B 0.000, C 0.000 }
gfCNCPoint3[12469] = {X 441.4171, Y 19.9718, Z -3.8333, A 0.000, B 0.000, C 0.000 }
gfCNCPoint3[12470] = {X 441.2703, Y 20.0647, Z -3.8333, A 0.000, B 0.000, C 0.000 }
gfCNCPoint3[12471] = {X 441.1809, Y 20.2136, Z -3.8333, A 0.000, B 0.000, C 0.000 }
gfCNCPoint3[12472] = {X 441.0209, Y 20.9600, Z -3.8333, A 0.000, B 0.000, C 0.000 }
gfCNCPoint3[12473] = {X 441.0072, Y 21.7232, Z -3.8333, A 0.000, B 0.000, C 0.000 }
gfCNCPoint3[12474] = {X 441.1404, Y 22.4749, Z -3.8333, A 0.000, B 0.000, C 0.000 }
gfCNCPoint3[12475] = {X 441.4297, Y 22.5608, Z -3.8333, A 0.000, B 0.000, C 0.000 }
gfCNCPoint3[12476] = {X 441.7277, Y 22.6079, Z -3.8333, A 0.000, B 0.000, C 0.000 }
gfCNCPoint3[12477] = {X 443.0590, Y 22.6957, Z -3.8333, A 0.000, B 0.000, C 0.000 }
gfCNCPoint3[12478] = {X 444.3930, Y 22.7160, Z -3.8333, A 0.000, B 0.000, C 0.000 }
gfCNCPoint3[12479] = {X 445.9287, Y 22.7160, Z -3.8333, A 0.000, B 0.000, C 0.000 }
gfCNCPoint3[12480] = {X 449.9135, Y 22.3674, Z -3.8333, A 0.000, B 0.000, C 0.000 }
gfCNCPoint3[12481] = {X 441.9439, Y 22.4474, Z -3.8333, A 0.000, B 0.000, C 0.000 }
gfCNCPoint3[12482] = {X 445.9287, Y 22.7960, Z -3.8333, A 0.000, B 0.000, C 0.000 }
gfCNCPoint3[12483] = {X 450.3584, Y 22.7960, Z -3.8333, A 0.000, B 0.000, C 0.000 }
gfCNCPoint3[12484] = {X 450.3584, Y 19.5417, Z -3.8333, A 0.000, B 0.000, C 0.000 }
gfCNCPoint3[12485] = {X 444.0385, Y 19.5414, Z -3.8333, A 0.000, B 0.000, C 0.000 }
gfCNCPoint3[12486] = {X 443.3470, Y 19.5576, Z -3.8333, A 0.000, B 0.000, C 0.000 }
gfCNCPoint3[12487] = {X 442.3555, Y 19.6485, Z -3.8333, A 0.000, B 0.000, C 0.000 }
gfCNCPoint3[12488] = {X 441.3911, Y 19.8961, Z -3.8333, A 0.000, B 0.000, C 0.000 }
gfCNCPoint3[12489] = {X 441.2131, Y 20.0088, Z -3.8333, A 0.000, B 0.000, C 0.000 }
gfCNCPoint3[12490] = {X 441.1046, Y 20.1894, Z -3.8333, A 0.000, B 0.000, C 0.000 }
gfCNCPoint3[12491] = {X 440.9399, Y 20.9643, Z -3.8333, A 0.000, B 0.000, C 0.000 }
gfCNCPoint3[12492] = {X 440.9297, Y 21.7565, Z -3.8333, A 0.000, B 0.000, C 0.000 }
gfCNCPoint3[12493] = {X 441.0745, Y 22.5354, Z -3.8333, A 0.000, B 0.000, C 0.000 }
gfCNCPoint3[12494] = {X 441.3921, Y 22.6342, Z -3.8333, A 0.000, B 0.000, C 0.000 }
gfCNCPoint3[12495] = {X 441.7204, Y 22.6876, Z -3.8333, A 0.000, B 0.000, C 0.000 }
gfCNCPoint3[12496] = {X 443.0556, Y 22.7756, Z -3.8333, A 0.000, B 0.000, C 0.000 }
gfCNCPoint3[12497] = {X 444.3934, Y 22.7960, Z -3.8333, A 0.000, B 0.000, C 0.000 }
gfCNCPoint3[12498] = {X 445.9287, Y 22.7960, Z -3.8333, A 0.000, B 0.000, C 0.000 }
gfCNCPoint3[12499] = {X 449.9135, Y 22.4474, Z -3.8333, A 0.000, B 0.000, C 0.000 }
gfCNCPoint3[12500] = {X 441.9439, Y 22.5274, Z -3.8333, A 0.000, B 0.000, C 0.000 }
gfCNCPoint3[12501] = {X 445.9287, Y 22.8760, Z -3.8333, A 0.000, B 0.000, C 0.000 }
gfCNCPoint3[12502] = {X 450.4384, Y 22.8760, Z -3.8333, A 0.000, B 0.000, C 0.000 }
gfCNCPoint3[12503] = {X 450.4384, Y 19.4617, Z -3.8333, A 0.000, B 0.000, C 0.000 }
gfCNCPoint3[12504] = {X 444.0376, Y 19.4614, Z -3.8333, A 0.000, B 0.000, C 0.000 }
gfCNCPoint3[12505] = {X 443.3456, Y 19.4776, Z -3.8333, A 0.000, B 0.000, C 0.000 }
gfCNCPoint3[12506] = {X 442.3416, Y 19.5697, Z -3.8333, A 0.000, B 0.000, C 0.000 }
gfCNCPoint3[12507] = {X 441.3651, Y 19.8205, Z -3.8333, A 0.000, B 0.000, C 0.000 }
gfCNCPoint3[12508] = {X 441.1558, Y 19.9529, Z -3.8333, A 0.000, B 0.000, C 0.000 }
gfCNCPoint3[12509] = {X 441.0284, Y 20.1651, Z -3.8333, A 0.000, B 0.000, C 0.000 }
gfCNCPoint3[12510] = {X 440.8589, Y 20.9684, Z -3.8333, A 0.000, B 0.000, C 0.000 }
gfCNCPoint3[12511] = {X 440.8523, Y 21.7894, Z -3.8333, A 0.000, B 0.000, C 0.000 }
gfCNCPoint3[12512] = {X 441.0087, Y 22.5953, Z -3.8333, A 0.000, B 0.000, C 0.000 }
gfCNCPoint3[12513] = {X 441.3545, Y 22.7075, Z -3.8333, A 0.000, B 0.000, C 0.000 }
gfCNCPoint3[12514] = {X 441.7131, Y 22.7673, Z -3.8333, A 0.000, B 0.000, C 0.000 }
gfCNCPoint3[12515] = {X 443.0521, Y 22.8555, Z -3.8333, A 0.000, B 0.000, C 0.000 }
gfCNCPoint3[12516] = {X 444.3938, Y 22.8760, Z -3.8333, A 0.000, B 0.000, C 0.000 }
gfCNCPoint3[12517] = {X 445.9287, Y 22.8760, Z -3.8333, A 0.000, B 0.000, C 0.000 }
gfCNCPoint3[12518] = {X 449.9135, Y 22.5274, Z -3.8333, A 0.000, B 0.000, C 0.000 }
gfCNCPoint3[12519] = {X 441.9439, Y 22.6074, Z -3.8333, A 0.000, B 0.000, C 0.000 }
gfCNCPoint3[12520] = {X 445.9287, Y 22.9560, Z -3.8333, A 0.000, B 0.000, C 0.000 }
gfCNCPoint3[12521] = {X 450.5184, Y 22.9560, Z -3.8333, A 0.000, B 0.000, C 0.000 }
gfCNCPoint3[12522] = {X 450.5192, Y 19.3817, Z -3.8333, A 0.000, B 0.000, C 0.000 }
gfCNCPoint3[12523] = {X 444.0367, Y 19.3814, Z -3.8333, A 0.000, B 0.000, C 0.000 }
gfCNCPoint3[12524] = {X 443.3442, Y 19.3977, Z -3.8333, A 0.000, B 0.000, C 0.000 }
gfCNCPoint3[12525] = {X 442.3277, Y 19.4909, Z -3.8333, A 0.000, B 0.000, C 0.000 }
gfCNCPoint3[12526] = {X 441.3390, Y 19.7448, Z -3.8333, A 0.000, B 0.000, C 0.000 }
gfCNCPoint3[12527] = {X 441.0986, Y 19.8970, Z -3.8333, A 0.000, B 0.000, C 0.000 }
gfCNCPoint3[12528] = {X 440.9522, Y 20.1409, Z -3.8333, A 0.000, B 0.000, C 0.000 }
gfCNCPoint3[12529] = {X 440.7780, Y 20.9724, Z -3.8333, A 0.000, B 0.000, C 0.000 }
gfCNCPoint3[12530] = {X 440.7750, Y 21.8219, Z -3.8333, A 0.000, B 0.000, C 0.000 }
gfCNCPoint3[12531] = {X 440.9432, Y 22.6546, Z -3.8333, A 0.000, B 0.000, C 0.000 }
gfCNCPoint3[12532] = {X 441.3170, Y 22.7806, Z -3.8333, A 0.000, B 0.000, C 0.000 }
gfCNCPoint3[12533] = {X 441.7059, Y 22.8469, Z -3.8333, A 0.000, B 0.000, C 0.000 }
gfCNCPoint3[12534] = {X 443.0487, Y 22.9354, Z -3.8333, A 0.000, B 0.000, C 0.000 }
gfCNCPoint3[12535] = {X 444.3942, Y 22.9560, Z -3.8333, A 0.000, B 0.000, C 0.000 }
gfCNCPoint3[12536] = {X 445.9287, Y 22.9560, Z -3.8333, A 0.000, B 0.000, C 0.000 }
gfCNCPoint3[12537] = {X 449.9135, Y 22.6074, Z -3.8333, A 0.000, B 0.000, C 0.000 }
gfCNCPoint3[12538] = {X 449.9135, Y 22.6074, Z -0.8333, A 0.000, B 0.000, C 0.000 }
gfCNCPoint3[12539] = {X 449.9135, Y 22.6074, Z 11.0000, A 0.000, B 0.000, C 0.000 }
gfCNCPoint3[12540] = {X 491.9901, Y 19.7814, Z 11.0000, A 0.000, B 0.000, C 0.000 }
gfCNCPoint3[12541] = {X 491.9901, Y 19.7814, Z 0.0000, A 0.000, B 0.000, C 0.000 }
gfCNCPoint3[12542] = {X 487.6645, Y 19.7807, Z -1.1590, A 0.000, B 0.000, C 0.000 }
gfCNCPoint3[12543] = {X 486.9699, Y 19.7855, Z -1.3452, A 0.000, B 0.000, C 0.000 }
gfCNCPoint3[12544] = {X 486.2675, Y 19.7841, Z -1.5334, A 0.000, B 0.000, C 0.000 }
gfCNCPoint3[12545] = {X 485.4760, Y 19.8890, Z -1.7473, A 0.000, B 0.000, C 0.000 }
gfCNCPoint3[12546] = {X 484.7983, Y 20.0734, Z -1.9355, A 0.000, B 0.000, C 0.000 }
gfCNCPoint3[12547] = {X 484.6641, Y 20.1100, Z -1.9728, A 0.000, B 0.000, C 0.000 }
gfCNCPoint3[12548] = {X 484.6325, Y 20.1397, Z -1.9844, A 0.000, B 0.000, C 0.000 }
gfCNCPoint3[12549] = {X 484.4392, Y 20.7097, Z -2.1457, A 0.000, B 0.000, C 0.000 }
gfCNCPoint3[12550] = {X 484.4040, Y 21.9085, Z -2.4670, A 0.000, B 0.000, C 0.000 }
gfCNCPoint3[12551] = {X 484.5267, Y 22.3547, Z -2.5910, A 0.000, B 0.000, C 0.000 }
gfCNCPoint3[12552] = {X 484.7217, Y 22.4182, Z -2.6460, A 0.000, B 0.000, C 0.000 }
gfCNCPoint3[12553] = {X 484.9351, Y 22.4359, Z -2.7033, A 0.000, B 0.000, C 0.000 }
gfCNCPoint3[12554] = {X 486.0892, Y 22.5573, Z -3.0143, A 0.000, B 0.000, C 0.000 }
gfCNCPoint3[12555] = {X 486.4781, Y 22.5746, Z -3.1186, A 0.000, B 0.000, C 0.000 }
gfCNCPoint3[12556] = {X 487.6448, Y 22.5560, Z -3.4312, A 0.000, B 0.000, C 0.000 }
gfCNCPoint3[12557] = {X 489.1454, Y 22.5560, Z -3.8333, A 0.000, B 0.000, C 0.000 }
gfCNCPoint3[12558] = {X 493.3690, Y 22.5560, Z -3.8333, A 0.000, B 0.000, C 0.000 }
gfCNCPoint3[12559] = {X 493.3690, Y 19.7816, Z -3.8333, A 0.000, B 0.000, C 0.000 }
gfCNCPoint3[12560] = {X 487.6645, Y 19.7807, Z -3.8333, A 0.000, B 0.000, C 0.000 }
gfCNCPoint3[12561] = {X 486.9699, Y 19.7855, Z -3.8333, A 0.000, B 0.000, C 0.000 }
gfCNCPoint3[12562] = {X 485.8745, Y 19.8567, Z -3.8333, A 0.000, B 0.000, C 0.000 }
gfCNCPoint3[12563] = {X 484.7983, Y 20.0734, Z -3.8333, A 0.000, B 0.000, C 0.000 }
gfCNCPoint3[12564] = {X 484.6684, Y 20.1462, Z -3.8333, A 0.000, B 0.000, C 0.000 }
gfCNCPoint3[12565] = {X 484.5878, Y 20.2714, Z -3.8333, A 0.000, B 0.000, C 0.000 }
gfCNCPoint3[12566] = {X 484.4289, Y 20.9572, Z -3.8333, A 0.000, B 0.000, C 0.000 }
gfCNCPoint3[12567] = {X 484.4083, Y 21.6608, Z -3.8333, A 0.000, B 0.000, C 0.000 }
gfCNCPoint3[12568] = {X 484.5267, Y 22.3547, Z -3.8333, A 0.000, B 0.000, C 0.000 }
gfCNCPoint3[12569] = {X 484.7285, Y 22.4074, Z -3.8333, A 0.000, B 0.000, C 0.000 }
gfCNCPoint3[12570] = {X 484.9351, Y 22.4359, Z -3.8333, A 0.000, B 0.000, C 0.000 }
gfCNCPoint3[12571] = {X 486.2881, Y 22.5370, Z -3.8333, A 0.000, B 0.000, C 0.000 }
gfCNCPoint3[12572] = {X 487.6448, Y 22.5560, Z -3.8333, A 0.000, B 0.000, C 0.000 }
gfCNCPoint3[12573] = {X 489.1454, Y 22.5560, Z -3.8333, A 0.000, B 0.000, C 0.000 }
gfCNCPoint3[12574] = {X 485.1606, Y 22.2874, Z -3.8333, A 0.000, B 0.000, C 0.000 }
gfCNCPoint3[12575] = {X 489.1454, Y 22.6360, Z -3.8333, A 0.000, B 0.000, C 0.000 }
gfCNCPoint3[12576] = {X 493.4490, Y 22.6360, Z -3.8333, A 0.000, B 0.000, C 0.000 }
gfCNCPoint3[12577] = {X 493.4490, Y 19.7016, Z -3.8333, A 0.000, B 0.000, C 0.000 }
gfCNCPoint3[12578] = {X 487.6642, Y 19.7007, Z -3.8333, A 0.000, B 0.000, C 0.000 }
gfCNCPoint3[12579] = {X 486.9714, Y 19.7055, Z -3.8333, A 0.000, B 0.000, C 0.000 }
gfCNCPoint3[12580] = {X 485.8646, Y 19.7773, Z -3.8333, A 0.000, B 0.000, C 0.000 }
gfCNCPoint3[12581] = {X 484.7773, Y 19.9962, Z -3.8333, A 0.000, B 0.000, C 0.000 }
gfCNCPoint3[12582] = {X 484.6136, Y 20.0879, Z -3.8333, A 0.000, B 0.000, C 0.000 }
gfCNCPoint3[12583] = {X 484.5121, Y 20.2457, Z -3.8333, A 0.000, B 0.000, C 0.000 }
gfCNCPoint3[12584] = {X 484.3478, Y 20.9610, Z -3.8333, A 0.000, B 0.000, C 0.000 }
gfCNCPoint3[12585] = {X 484.3306, Y 21.6947, Z -3.8333, A 0.000, B 0.000, C 0.000 }
gfCNCPoint3[12586] = {X 484.4611, Y 22.4170, Z -3.8333, A 0.000, B 0.000, C 0.000 }
gfCNCPoint3[12587] = {X 484.6880, Y 22.4807, Z -3.8333, A 0.000, B 0.000, C 0.000 }
gfCNCPoint3[12588] = {X 484.9212, Y 22.5149, Z -3.8333, A 0.000, B 0.000, C 0.000 }
gfCNCPoint3[12589] = {X 486.2799, Y 22.6167, Z -3.8333, A 0.000, B 0.000, C 0.000 }
gfCNCPoint3[12590] = {X 487.6422, Y 22.6360, Z -3.8333, A 0.000, B 0.000, C 0.000 }
gfCNCPoint3[12591] = {X 489.1454, Y 22.6360, Z -3.8333, A 0.000, B 0.000, C 0.000 }
gfCNCPoint3[12592] = {X 493.1302, Y 22.2874, Z -3.8333, A 0.000, B 0.000, C 0.000 }
gfCNCPoint3[12593] = {X 485.1606, Y 22.3674, Z -3.8333, A 0.000, B 0.000, C 0.000 }
gfCNCPoint3[12594] = {X 489.1454, Y 22.7160, Z -3.8333, A 0.000, B 0.000, C 0.000 }
gfCNCPoint3[12595] = {X 493.5290, Y 22.7160, Z -3.8333, A 0.000, B 0.000, C 0.000 }
gfCNCPoint3[12596] = {X 493.5290, Y 19.6216, Z -3.8333, A 0.000, B 0.000, C 0.000 }
gfCNCPoint3[12597] = {X 487.6640, Y 19.6207, Z -3.8333, A 0.000, B 0.000, C 0.000 }
gfCNCPoint3[12598] = {X 486.9712, Y 19.6255, Z -3.8333, A 0.000, B 0.000, C 0.000 }
gfCNCPoint3[12599] = {X 485.8539, Y 19.6980, Z -3.8333, A 0.000, B 0.000, C 0.000 }
gfCNCPoint3[12600] = {X 484.7563, Y 19.9190, Z -3.8333, A 0.000, B 0.000, C 0.000 }
gfCNCPoint3[12601] = {X 484.5588, Y 20.0296, Z -3.8333, A 0.000, B 0.000, C 0.000 }
gfCNCPoint3[12602] = {X 484.4363, Y 20.2201, Z -3.8333, A 0.000, B 0.000, C 0.000 }
gfCNCPoint3[12603] = {X 484.2668, Y 20.9646, Z -3.8333, A 0.000, B 0.000, C 0.000 }
gfCNCPoint3[12604] = {X 484.2530, Y 21.7281, Z -3.8333, A 0.000, B 0.000, C 0.000 }
gfCNCPoint3[12605] = {X 484.3957, Y 22.4783, Z -3.8333, A 0.000, B 0.000, C 0.000 }
gfCNCPoint3[12606] = {X 484.6512, Y 22.5545, Z -3.8333, A 0.000, B 0.000, C 0.000 }
gfCNCPoint3[12607] = {X 484.9147, Y 22.5947, Z -3.8333, A 0.000, B 0.000, C 0.000 }
gfCNCPoint3[12608] = {X 486.2770, Y 22.6966, Z -3.8333, A 0.000, B 0.000, C 0.000 }
gfCNCPoint3[12609] = {X 487.6429, Y 22.7160, Z -3.8333, A 0.000, B 0.000, C 0.000 }
gfCNCPoint3[12610] = {X 489.1454, Y 22.7160, Z -3.8333, A 0.000, B 0.000, C 0.000 }
gfCNCPoint3[12611] = {X 493.1302, Y 22.3674, Z -3.8333, A 0.000, B 0.000, C 0.000 }
gfCNCPoint3[12612] = {X 485.1606, Y 22.4474, Z -3.8333, A 0.000, B 0.000, C 0.000 }
gfCNCPoint3[12613] = {X 489.1454, Y 22.7960, Z -3.8333, A 0.000, B 0.000, C 0.000 }
gfCNCPoint3[12614] = {X 493.6090, Y 22.7960, Z -3.8333, A 0.000, B 0.000, C 0.000 }
gfCNCPoint3[12615] = {X 493.6090, Y 19.5417, Z -3.8333, A 0.000, B 0.000, C 0.000 }
gfCNCPoint3[12616] = {X 487.6637, Y 19.5407, Z -3.8333, A 0.000, B 0.000, C 0.000 }
gfCNCPoint3[12617] = {X 486.9711, Y 19.5455, Z -3.8333, A 0.000, B 0.000, C 0.000 }
gfCNCPoint3[12618] = {X 485.8433, Y 19.6187, Z -3.8333, A 0.000, B 0.000, C 0.000 }
gfCNCPoint3[12619] = {X 484.7353, Y 19.8419, Z -3.8333, A 0.000, B 0.000, C 0.000 }
gfCNCPoint3[12620] = {X 484.5040, Y 19.9713, Z -3.8333, A 0.000, B 0.000, C 0.000 }
gfCNCPoint3[12621] = {X 484.3606, Y 20.1944, Z -3.8333, A 0.000, B 0.000, C 0.000 }
gfCNCPoint3[12622] = {X 484.1858, Y 20.9680, Z -3.8333, A 0.000, B 0.000, C 0.000 }
gfCNCPoint3[12623] = {X 484.1756, Y 21.7610, Z -3.8333, A 0.000, B 0.000, C 0.000 }
gfCNCPoint3[12624] = {X 484.3305, Y 22.5389, Z -3.8333, A 0.000, B 0.000, C 0.000 }
gfCNCPoint3[12625] = {X 484.6139, Y 22.6281, Z -3.8333, A 0.000, B 0.000, C 0.000 }
gfCNCPoint3[12626] = {X 484.9073, Y 22.6743, Z -3.8333, A 0.000, B 0.000, C 0.000 }
gfCNCPoint3[12627] = {X 486.2736, Y 22.7765, Z -3.8333, A 0.000, B 0.000, C 0.000 }
gfCNCPoint3[12628] = {X 487.6435, Y 22.7960, Z -3.8333, A 0.000, B 0.000, C 0.000 }
gfCNCPoint3[12629] = {X 489.1454, Y 22.7960, Z -3.8333, A 0.000, B 0.000, C 0.000 }
gfCNCPoint3[12630] = {X 493.1302, Y 22.4474, Z -3.8333, A 0.000, B 0.000, C 0.000 }
gfCNCPoint3[12631] = {X 485.1606, Y 22.5274, Z -3.8333, A 0.000, B 0.000, C 0.000 }
gfCNCPoint3[12632] = {X 489.1454, Y 22.8760, Z -3.8333, A 0.000, B 0.000, C 0.000 }
gfCNCPoint3[12633] = {X 493.6890, Y 22.8760, Z -3.8333, A 0.000, B 0.000, C 0.000 }
gfCNCPoint3[12634] = {X 493.6890, Y 19.4617, Z -3.8333, A 0.000, B 0.000, C 0.000 }
gfCNCPoint3[12635] = {X 487.6634, Y 19.4607, Z -3.8333, A 0.000, B 0.000, C 0.000 }
gfCNCPoint3[12636] = {X 486.9709, Y 19.4655, Z -3.8333, A 0.000, B 0.000, C 0.000 }
gfCNCPoint3[12637] = {X 485.8326, Y 19.5394, Z -3.8333, A 0.000, B 0.000, C 0.000 }
gfCNCPoint3[12638] = {X 484.7143, Y 19.7647, Z -3.8333, A 0.000, B 0.000, C 0.000 }
gfCNCPoint3[12639] = {X 484.4491, Y 19.9131, Z -3.8333, A 0.000, B 0.000, C 0.000 }
gfCNCPoint3[12640] = {X 484.2848, Y 20.1687, Z -3.8333, A 0.000, B 0.000, C 0.000 }
gfCNCPoint3[12641] = {X 484.1049, Y 20.9711, Z -3.8333, A 0.000, B 0.000, C 0.000 }
gfCNCPoint3[12642] = {X 484.0984, Y 21.7935, Z -3.8333, A 0.000, B 0.000, C 0.000 }
gfCNCPoint3[12643] = {X 484.2656, Y 22.5987, Z -3.8333, A 0.000, B 0.000, C 0.000 }
gfCNCPoint3[12644] = {X 484.5765, Y 22.7014, Z -3.8333, A 0.000, B 0.000, C 0.000 }
gfCNCPoint3[12645] = {X 484.8998, Y 22.7540, Z -3.8333, A 0.000, B 0.000, C 0.000 }
gfCNCPoint3[12646] = {X 486.2701, Y 22.8565, Z -3.8333, A 0.000, B 0.000, C 0.000 }
gfCNCPoint3[12647] = {X 487.6442, Y 22.8760, Z -3.8333, A 0.000, B 0.000, C 0.000 }
gfCNCPoint3[12648] = {X 489.1454, Y 22.8760, Z -3.8333, A 0.000, B 0.000, C 0.000 }
gfCNCPoint3[12649] = {X 493.1302, Y 22.5274, Z -3.8333, A 0.000, B 0.000, C 0.000 }
gfCNCPoint3[12650] = {X 485.1606, Y 22.6074, Z -3.8333, A 0.000, B 0.000, C 0.000 }
gfCNCPoint3[12651] = {X 489.1454, Y 22.9560, Z -3.8333, A 0.000, B 0.000, C 0.000 }
gfCNCPoint3[12652] = {X 493.7690, Y 22.9560, Z -3.8333, A 0.000, B 0.000, C 0.000 }
gfCNCPoint3[12653] = {X 493.7697, Y 19.3817, Z -3.8333, A 0.000, B 0.000, C 0.000 }
gfCNCPoint3[12654] = {X 487.6632, Y 19.3807, Z -3.8333, A 0.000, B 0.000, C 0.000 }
gfCNCPoint3[12655] = {X 486.9707, Y 19.3855, Z -3.8333, A 0.000, B 0.000, C 0.000 }
gfCNCPoint3[12656] = {X 485.8219, Y 19.4601, Z -3.8333, A 0.000, B 0.000, C 0.000 }
gfCNCPoint3[12657] = {X 484.6933, Y 19.6875, Z -3.8333, A 0.000, B 0.000, C 0.000 }
gfCNCPoint3[12658] = {X 484.3943, Y 19.8548, Z -3.8333, A 0.000, B 0.000, C 0.000 }
gfCNCPoint3[12659] = {X 484.2090, Y 20.1430, Z -3.8333, A 0.000, B 0.000, C 0.000 }
gfCNCPoint3[12660] = {X 484.0240, Y 20.9741, Z -3.8333, A 0.000, B 0.000, C 0.000 }
gfCNCPoint3[12661] = {X 484.0212, Y 21.8256, Z -3.8333, A 0.000, B 0.000, C 0.000 }
gfCNCPoint3[12662] = {X 484.2007, Y 22.6579, Z -3.8333, A 0.000, B 0.000, C 0.000 }
gfCNCPoint3[12663] = {X 484.5397, Y 22.7746, Z -3.8333, A 0.000, B 0.000, C 0.000 }
gfCNCPoint3[12664] = {X 484.8932, Y 22.8337, Z -3.8333, A 0.000, B 0.000, C 0.000 }
gfCNCPoint3[12665] = {X 486.2672, Y 22.9364, Z -3.8333, A 0.000, B 0.000, C 0.000 }
gfCNCPoint3[12666] = {X 487.6448, Y 22.9560, Z -3.8333, A 0.000, B 0.000, C 0.000 }
gfCNCPoint3[12667] = {X 489.1454, Y 22.9560, Z -3.8333, A 0.000, B 0.000, C 0.000 }
gfCNCPoint3[12668] = {X 493.1302, Y 22.6074, Z -3.8333, A 0.000, B 0.000, C 0.000 }
gfCNCPoint3[12669] = {X 493.1302, Y 22.6074, Z -0.8333, A 0.000, B 0.000, C 0.000 }
gfCNCPoint3[12670] = {X 493.1302, Y 22.6074, Z 11.0000, A 0.000, B 0.000, C 0.000 }
gfCNCPoint3[12671] = {X 607.6965, Y 2.1249, Z 11.0000, A 0.000, B 0.000, C 0.000 }
gfCNCPoint3[12672] = {X 607.6965, Y 2.1249, Z -0.8333, A 0.000, B 0.000, C 0.000 }
gfCNCPoint3[12673] = {X 607.6965, Y 2.1249, Z -3.8333, A 0.000, B 0.000, C 0.000 }
gfCNCPoint3[12674] = {X 603.6965, Y 8.3206, Z -3.8333, A 0.000, B 0.000, C 0.000 }
gfCNCPoint3[12675] = {X 603.3204, Y 8.8211, Z -3.8333, A 0.000, B 0.000, C 0.000 }
gfCNCPoint3[12676] = {X 602.8770, Y 9.2631, Z -3.8333, A 0.000, B 0.000, C 0.000 }
gfCNCPoint3[12677] = {X 602.8769, Y 40.7368, Z -3.8333, A 0.000, B 0.000, C 0.000 }
gfCNCPoint3[12678] = {X 603.3204, Y 41.1789, Z -3.8333, A 0.000, B 0.000, C 0.000 }
gfCNCPoint3[12679] = {X 603.6965, Y 41.6794, Z -3.8333, A 0.000, B 0.000, C 0.000 }
gfCNCPoint3[12680] = {X 607.6965, Y 47.8751, Z -3.8333, A 0.000, B 0.000, C 0.000 }
gfCNCPoint3[12681] = {X 607.6965, Y 47.8751, Z -0.8333, A 0.000, B 0.000, C 0.000 }
gfCNCPoint3[12682] = {X 607.6965, Y 47.8751, Z 11.0000, A 0.000, B 0.000, C 0.000 }
gfCNCPoint3[12683] = {X 607.6965, Y 1.5491, Z 11.0000, A 0.000, B 0.000, C 0.000 }
gfCNCPoint3[12684] = {X 607.6965, Y 1.5491, Z -0.8333, A 0.000, B 0.000, C 0.000 }
gfCNCPoint3[12685] = {X 607.6965, Y 1.5491, Z -3.8333, A 0.000, B 0.000, C 0.000 }
gfCNCPoint3[12686] = {X 603.6965, Y 8.1705, Z -3.8333, A 0.000, B 0.000, C 0.000 }
gfCNCPoint3[12687] = {X 603.2896, Y 8.7357, Z -3.8333, A 0.000, B 0.000, C 0.000 }
gfCNCPoint3[12688] = {X 602.7970, Y 9.2281, Z -3.8333, A 0.000, B 0.000, C 0.000 }
gfCNCPoint3[12689] = {X 602.7969, Y 40.7725, Z -3.8333, A 0.000, B 0.000, C 0.000 }
gfCNCPoint3[12690] = {X 603.2895, Y 41.2648, Z -3.8333, A 0.000, B 0.000, C 0.000 }
gfCNCPoint3[12691] = {X 603.6965, Y 41.8298, Z -3.8333, A 0.000, B 0.000, C 0.000 }
gfCNCPoint3[12692] = {X 607.6965, Y 48.4482, Z -3.8333, A 0.000, B 0.000, C 0.000 }
gfCNCPoint3[12693] = {X 607.6965, Y 48.4482, Z -0.8333, A 0.000, B 0.000, C 0.000 }
gfCNCPoint3[12694] = {X 607.6965, Y 48.4482, Z 11.0000, A 0.000, B 0.000, C 0.000 }
gfCNCPoint3[12695] = {X 607.6965, Y 0.8830, Z 11.0000, A 0.000, B 0.000, C 0.000 }
gfCNCPoint3[12696] = {X 607.6965, Y 0.8830, Z -0.8333, A 0.000, B 0.000, C 0.000 }
gfCNCPoint3[12697] = {X 607.6965, Y 0.8830, Z -3.8333, A 0.000, B 0.000, C 0.000 }
gfCNCPoint3[12698] = {X 603.6965, Y 8.0116, Z -3.8333, A 0.000, B 0.000, C 0.000 }
gfCNCPoint3[12699] = {X 603.2605, Y 8.6459, Z -3.8333, A 0.000, B 0.000, C 0.000 }
gfCNCPoint3[12700] = {X 602.7170, Y 9.1909, Z -3.8333, A 0.000, B 0.000, C 0.000 }
gfCNCPoint3[12701] = {X 602.7169, Y 40.8098, Z -3.8333, A 0.000, B 0.000, C 0.000 }
gfCNCPoint3[12702] = {X 603.2605, Y 41.3546, Z -3.8333, A 0.000, B 0.000, C 0.000 }
gfCNCPoint3[12703] = {X 603.6965, Y 41.9887, Z -3.8333, A 0.000, B 0.000, C 0.000 }
gfCNCPoint3[12704] = {X 607.6965, Y 49.1137, Z -3.8333, A 0.000, B 0.000, C 0.000 }
gfCNCPoint3[12705] = {X 607.6965, Y 49.1137, Z -0.8333, A 0.000, B 0.000, C 0.000 }
gfCNCPoint3[12706] = {X 607.6965, Y 49.1137, Z 11.0000, A 0.000, B 0.000, C 0.000 }
gfCNCPoint3[12707] = {X 607.6950, Y 0.0857, Z 11.0000, A 0.000, B 0.000, C 0.000 }
gfCNCPoint3[12708] = {X 607.6950, Y 0.0857, Z -0.8333, A 0.000, B 0.000, C 0.000 }
gfCNCPoint3[12709] = {X 607.6950, Y 0.0857, Z -3.8333, A 0.000, B 0.000, C 0.000 }
gfCNCPoint3[12710] = {X 603.6965, Y 7.8428, Z -3.8333, A 0.000, B 0.000, C 0.000 }
gfCNCPoint3[12711] = {X 603.2338, Y 8.5522, Z -3.8333, A 0.000, B 0.000, C 0.000 }
gfCNCPoint3[12712] = {X 602.6370, Y 9.1532, Z -3.8333, A 0.000, B 0.000, C 0.000 }
gfCNCPoint3[12713] = {X 602.6369, Y 40.8474, Z -3.8333, A 0.000, B 0.000, C 0.000 }
gfCNCPoint3[12714] = {X 603.2338, Y 41.4482, Z -3.8333, A 0.000, B 0.000, C 0.000 }
gfCNCPoint3[12715] = {X 603.6965, Y 42.1574, Z -3.8333, A 0.000, B 0.000, C 0.000 }
gfCNCPoint3[12716] = {X 607.6965, Y 49.9129, Z -3.8333, A 0.000, B 0.000, C 0.000 }
gfCNCPoint3[12717] = {X 607.6965, Y 49.9129, Z -0.8333, A 0.000, B 0.000, C 0.000 }
gfCNCPoint3[12718] = {X 607.6965, Y 49.9129, Z 11.0000, A 0.000, B 0.000, C 0.000 }
gfCNCPoint3[12719] = {X 607.6538, Y -0.8102, Z 11.0000, A 0.000, B 0.000, C 0.000 }
gfCNCPoint3[12720] = {X 607.6538, Y -0.8102, Z -0.8333, A 0.000, B 0.000, C 0.000 }
gfCNCPoint3[12721] = {X 607.6538, Y -0.8102, Z -3.8333, A 0.000, B 0.000, C 0.000 }
gfCNCPoint3[12722] = {X 603.6965, Y 7.6609, Z -3.8333, A 0.000, B 0.000, C 0.000 }
gfCNCPoint3[12723] = {X 603.2070, Y 8.4562, Z -3.8333, A 0.000, B 0.000, C 0.000 }
gfCNCPoint3[12724] = {X 602.5495, Y 9.1194, Z -3.8333, A 0.000, B 0.000, C 0.000 }
gfCNCPoint3[12725] = {X 602.5570, Y 9.1532, Z -3.8333, A 0.000, B 0.000, C 0.000 }
gfCNCPoint3[12726] = {X 602.5569, Y 40.8855, Z -3.8333, A 0.000, B 0.000, C 0.000 }
gfCNCPoint3[12727] = {X 603.2101, Y 41.5469, Z -3.8333, A 0.000, B 0.000, C 0.000 }
gfCNCPoint3[12728] = {X 603.6965, Y 42.3389, Z -3.8333, A 0.000, B 0.000, C 0.000 }
gfCNCPoint3[12729] = {X 607.6965, Y 50.9101, Z -3.8333, A 0.000, B 0.000, C 0.000 }
gfCNCPoint3[12730] = {X 607.6965, Y 50.9101, Z -0.8333, A 0.000, B 0.000, C 0.000 }
gfCNCPoint3[12731] = {X 607.6965, Y 50.9101, Z 11.0000, A 0.000, B 0.000, C 0.000 }
gfCNCPoint3[12732] = {X 607.4987, Y -1.7344, Z 11.0000, A 0.000, B 0.000, C 0.000 }
gfCNCPoint3[12733] = {X 607.4987, Y -1.7344, Z -0.8333, A 0.000, B 0.000, C 0.000 }
gfCNCPoint3[12734] = {X 607.4987, Y -1.7344, Z -3.8333, A 0.000, B 0.000, C 0.000 }
gfCNCPoint3[12735] = {X 603.6965, Y 7.4623, Z -3.8333, A 0.000, B 0.000, C 0.000 }
gfCNCPoint3[12736] = {X 603.3769, Y 8.0781, Z -3.8333, A 0.000, B 0.000, C 0.000 }
gfCNCPoint3[12737] = {X 602.9556, Y 8.6293, Z -3.8333, A 0.000, B 0.000, C 0.000 }
gfCNCPoint3[12738] = {X 602.4454, Y 9.0995, Z -3.8333, A 0.000, B 0.000, C 0.000 }
gfCNCPoint3[12739] = {X 602.4770, Y 9.1532, Z -3.8333, A 0.000, B 0.000, C 0.000 }
gfCNCPoint3[12740] = {X 602.4769, Y 40.9228, Z -3.8333, A 0.000, B 0.000, C 0.000 }
gfCNCPoint3[12741] = {X 602.5727, Y 41.0031, Z -3.8333, A 0.000, B 0.000, C 0.000 }
gfCNCPoint3[12742] = {X 603.2272, Y 41.7026, Z -3.8333, A 0.000, B 0.000, C 0.000 }
gfCNCPoint3[12743] = {X 603.6965, Y 42.5377, Z -3.8333, A 0.000, B 0.000, C 0.000 }
gfCNCPoint3[12744] = {X 607.6965, Y 52.2129, Z -3.8333, A 0.000, B 0.000, C 0.000 }
gfCNCPoint3[12745] = {X 607.6965, Y 52.2129, Z -0.8333, A 0.000, B 0.000, C 0.000 }
gfCNCPoint3[12746] = {X 607.6965, Y 52.2129, Z 11.0000, A 0.000, B 0.000, C 0.000 }
gfCNCPoint3[12747] = {X 607.6966, Y 2.1247, Z 11.0000, A 0.000, B 0.000, C 0.000 }
gfCNCPoint3[12748] = {X 607.6966, Y 2.1247, Z -1.6667, A 0.000, B 0.000, C 0.000 }
gfCNCPoint3[12749] = {X 607.6966, Y 2.1247, Z -4.6667, A 0.000, B 0.000, C 0.000 }
gfCNCPoint3[12750] = {X 603.6966, Y 8.3206, Z -4.6667, A 0.000, B 0.000, C 0.000 }
gfCNCPoint3[12751] = {X 603.3206, Y 8.8209, Z -4.6667, A 0.000, B 0.000, C 0.000 }
gfCNCPoint3[12752] = {X 602.8774, Y 9.2628, Z -4.6667, A 0.000, B 0.000, C 0.000 }
gfCNCPoint3[12753] = {X 602.8772, Y 40.7371, Z -4.6667, A 0.000, B 0.000, C 0.000 }
gfCNCPoint3[12754] = {X 603.3205, Y 41.1790, Z -4.6667, A 0.000, B 0.000, C 0.000 }
gfCNCPoint3[12755] = {X 603.6966, Y 41.6794, Z -4.6667, A 0.000, B 0.000, C 0.000 }
gfCNCPoint3[12756] = {X 607.6966, Y 47.8753, Z -4.6667, A 0.000, B 0.000, C 0.000 }
gfCNCPoint3[12757] = {X 607.6966, Y 47.8753, Z -1.6667, A 0.000, B 0.000, C 0.000 }
gfCNCPoint3[12758] = {X 607.6966, Y 47.8753, Z 11.0000, A 0.000, B 0.000, C 0.000 }
gfCNCPoint3[12759] = {X 607.6966, Y 1.5479, Z 11.0000, A 0.000, B 0.000, C 0.000 }
gfCNCPoint3[12760] = {X 607.6966, Y 1.5479, Z -1.6667, A 0.000, B 0.000, C 0.000 }
gfCNCPoint3[12761] = {X 607.6966, Y 1.5479, Z -4.6667, A 0.000, B 0.000, C 0.000 }
gfCNCPoint3[12762] = {X 603.6966, Y 8.1706, Z -4.6667, A 0.000, B 0.000, C 0.000 }
gfCNCPoint3[12763] = {X 603.2897, Y 8.7357, Z -4.6667, A 0.000, B 0.000, C 0.000 }
gfCNCPoint3[12764] = {X 602.7974, Y 9.2281, Z -4.6667, A 0.000, B 0.000, C 0.000 }
gfCNCPoint3[12765] = {X 602.7972, Y 40.7725, Z -4.6667, A 0.000, B 0.000, C 0.000 }
gfCNCPoint3[12766] = {X 603.2896, Y 41.2648, Z -4.6667, A 0.000, B 0.000, C 0.000 }
gfCNCPoint3[12767] = {X 603.6966, Y 41.8297, Z -4.6667, A 0.000, B 0.000, C 0.000 }
gfCNCPoint3[12768] = {X 607.6966, Y 48.4494, Z -4.6667, A 0.000, B 0.000, C 0.000 }
gfCNCPoint3[12769] = {X 607.6966, Y 48.4494, Z -1.6667, A 0.000, B 0.000, C 0.000 }
gfCNCPoint3[12770] = {X 607.6966, Y 48.4494, Z 11.0000, A 0.000, B 0.000, C 0.000 }
gfCNCPoint3[12771] = {X 607.6966, Y 0.8814, Z 11.0000, A 0.000, B 0.000, C 0.000 }
gfCNCPoint3[12772] = {X 607.6966, Y 0.8814, Z -1.6667, A 0.000, B 0.000, C 0.000 }
gfCNCPoint3[12773] = {X 607.6966, Y 0.8814, Z -4.6667, A 0.000, B 0.000, C 0.000 }
gfCNCPoint3[12774] = {X 603.6966, Y 8.0116, Z -4.6667, A 0.000, B 0.000, C 0.000 }
gfCNCPoint3[12775] = {X 603.2607, Y 8.6459, Z -4.6667, A 0.000, B 0.000, C 0.000 }
gfCNCPoint3[12776] = {X 602.7174, Y 9.1909, Z -4.6667, A 0.000, B 0.000, C 0.000 }
gfCNCPoint3[12777] = {X 602.7172, Y 40.8097, Z -4.6667, A 0.000, B 0.000, C 0.000 }
gfCNCPoint3[12778] = {X 603.2606, Y 41.3546, Z -4.6667, A 0.000, B 0.000, C 0.000 }
gfCNCPoint3[12779] = {X 603.6966, Y 41.9886, Z -4.6667, A 0.000, B 0.000, C 0.000 }
gfCNCPoint3[12780] = {X 607.6966, Y 49.1152, Z -4.6667, A 0.000, B 0.000, C 0.000 }
gfCNCPoint3[12781] = {X 607.6966, Y 49.1152, Z -1.6667, A 0.000, B 0.000, C 0.000 }
gfCNCPoint3[12782] = {X 607.6966, Y 49.1152, Z 11.0000, A 0.000, B 0.000, C 0.000 }
gfCNCPoint3[12783] = {X 607.6951, Y 0.0837, Z 11.0000, A 0.000, B 0.000, C 0.000 }
gfCNCPoint3[12784] = {X 607.6951, Y 0.0837, Z -1.6667, A 0.000, B 0.000, C 0.000 }
gfCNCPoint3[12785] = {X 607.6951, Y 0.0837, Z -4.6667, A 0.000, B 0.000, C 0.000 }
gfCNCPoint3[12786] = {X 603.6966, Y 7.8428, Z -4.6667, A 0.000, B 0.000, C 0.000 }
gfCNCPoint3[12787] = {X 603.2340, Y 8.5522, Z -4.6667, A 0.000, B 0.000, C 0.000 }
gfCNCPoint3[12788] = {X 602.6374, Y 9.1532, Z -4.6667, A 0.000, B 0.000, C 0.000 }
gfCNCPoint3[12789] = {X 602.6372, Y 40.8474, Z -4.6667, A 0.000, B 0.000, C 0.000 }
gfCNCPoint3[12790] = {X 603.2339, Y 41.4482, Z -4.6667, A 0.000, B 0.000, C 0.000 }
gfCNCPoint3[12791] = {X 603.6966, Y 42.1574, Z -4.6667, A 0.000, B 0.000, C 0.000 }
gfCNCPoint3[12792] = {X 607.6966, Y 49.9148, Z -4.6667, A 0.000, B 0.000, C 0.000 }
gfCNCPoint3[12793] = {X 607.6966, Y 49.9148, Z -1.6667, A 0.000, B 0.000, C 0.000 }
gfCNCPoint3[12794] = {X 607.6966, Y 49.9148, Z 11.0000, A 0.000, B 0.000, C 0.000 }
gfCNCPoint3[12795] = {X 607.6538, Y -0.8106, Z 11.0000, A 0.000, B 0.000, C 0.000 }
gfCNCPoint3[12796] = {X 607.6538, Y -0.8106, Z -1.6667, A 0.000, B 0.000, C 0.000 }
gfCNCPoint3[12797] = {X 607.6538, Y -0.8106, Z -4.6667, A 0.000, B 0.000, C 0.000 }
gfCNCPoint3[12798] = {X 603.6966, Y 7.6608, Z -4.6667, A 0.000, B 0.000, C 0.000 }
gfCNCPoint3[12799] = {X 603.2072, Y 8.4561, Z -4.6667, A 0.000, B 0.000, C 0.000 }
gfCNCPoint3[12800] = {X 602.5498, Y 9.1192, Z -4.6667, A 0.000, B 0.000, C 0.000 }
gfCNCPoint3[12801] = {X 602.5574, Y 9.1532, Z -4.6667, A 0.000, B 0.000, C 0.000 }
gfCNCPoint3[12802] = {X 602.5572, Y 40.8855, Z -4.6667, A 0.000, B 0.000, C 0.000 }
gfCNCPoint3[12803] = {X 603.2102, Y 41.5469, Z -4.6667, A 0.000, B 0.000, C 0.000 }
gfCNCPoint3[12804] = {X 603.6966, Y 42.3389, Z -4.6667, A 0.000, B 0.000, C 0.000 }
gfCNCPoint3[12805] = {X 607.6966, Y 50.9127, Z -4.6667, A 0.000, B 0.000, C 0.000 }
gfCNCPoint3[12806] = {X 607.6966, Y 50.9127, Z -1.6667, A 0.000, B 0.000, C 0.000 }
gfCNCPoint3[12807] = {X 607.6966, Y 50.9127, Z 11.0000, A 0.000, B 0.000, C 0.000 }
gfCNCPoint3[12808] = {X 607.4987, Y -1.7348, Z 11.0000, A 0.000, B 0.000, C 0.000 }
gfCNCPoint3[12809] = {X 607.4987, Y -1.7348, Z -1.6667, A 0.000, B 0.000, C 0.000 }
gfCNCPoint3[12810] = {X 607.4987, Y -1.7348, Z -4.6667, A 0.000, B 0.000, C 0.000 }
gfCNCPoint3[12811] = {X 603.6966, Y 7.4622, Z -4.6667, A 0.000, B 0.000, C 0.000 }
gfCNCPoint3[12812] = {X 603.3769, Y 8.0780, Z -4.6667, A 0.000, B 0.000, C 0.000 }
gfCNCPoint3[12813] = {X 602.9556, Y 8.6293, Z -4.6667, A 0.000, B 0.000, C 0.000 }
gfCNCPoint3[12814] = {X 602.4454, Y 9.0995, Z -4.6667, A 0.000, B 0.000, C 0.000 }
gfCNCPoint3[12815] = {X 602.4774, Y 9.1532, Z -4.6667, A 0.000, B 0.000, C 0.000 }
gfCNCPoint3[12816] = {X 602.4772, Y 40.9227, Z -4.6667, A 0.000, B 0.000, C 0.000 }
gfCNCPoint3[12817] = {X 602.5728, Y 41.0031, Z -4.6667, A 0.000, B 0.000, C 0.000 }
gfCNCPoint3[12818] = {X 603.2272, Y 41.7027, Z -4.6667, A 0.000, B 0.000, C 0.000 }
gfCNCPoint3[12819] = {X 603.6966, Y 42.5378, Z -4.6667, A 0.000, B 0.000, C 0.000 }
gfCNCPoint3[12820] = {X 607.6966, Y 52.2135, Z -4.6667, A 0.000, B 0.000, C 0.000 }
gfCNCPoint3[12821] = {X 607.6966, Y 52.2135, Z -1.6667, A 0.000, B 0.000, C 0.000 }
gfCNCPoint3[12822] = {X 607.6966, Y 52.2135, Z 11.0000, A 0.000, B 0.000, C 0.000 }
gfCNCPoint3[12823] = {X 491.9911, Y 19.7817, Z 11.0000, A 0.000, B 0.000, C 0.000 }
gfCNCPoint3[12824] = {X 491.9911, Y 19.7817, Z -0.8333, A 0.000, B 0.000, C 0.000 }
gfCNCPoint3[12825] = {X 487.6645, Y 19.7811, Z -1.9926, A 0.000, B 0.000, C 0.000 }
gfCNCPoint3[12826] = {X 486.9699, Y 19.7858, Z -2.1788, A 0.000, B 0.000, C 0.000 }
gfCNCPoint3[12827] = {X 486.2675, Y 19.7844, Z -2.3670, A 0.000, B 0.000, C 0.000 }
gfCNCPoint3[12828] = {X 485.4763, Y 19.8893, Z -2.5808, A 0.000, B 0.000, C 0.000 }
gfCNCPoint3[12829] = {X 484.7986, Y 20.0737, Z -2.7690, A 0.000, B 0.000, C 0.000 }
gfCNCPoint3[12830] = {X 484.6643, Y 20.1102, Z -2.8063, A 0.000, B 0.000, C 0.000 }
gfCNCPoint3[12831] = {X 484.6322, Y 20.1405, Z -2.8181, A 0.000, B 0.000, C 0.000 }
gfCNCPoint3[12832] = {X 484.5876, Y 20.2724, Z -2.8554, A 0.000, B 0.000, C 0.000 }
gfCNCPoint3[12833] = {X 484.4393, Y 20.7113, Z -2.9796, A 0.000, B 0.000, C 0.000 }
gfCNCPoint3[12834] = {X 484.4044, Y 21.9076, Z -3.3003, A 0.000, B 0.000, C 0.000 }
gfCNCPoint3[12835] = {X 484.5268, Y 22.3544, Z -3.4244, A 0.000, B 0.000, C 0.000 }
gfCNCPoint3[12836] = {X 484.7218, Y 22.4178, Z -3.4793, A 0.000, B 0.000, C 0.000 }
gfCNCPoint3[12837] = {X 484.9348, Y 22.4355, Z -3.5366, A 0.000, B 0.000, C 0.000 }
gfCNCPoint3[12838] = {X 486.0968, Y 22.5570, Z -3.8497, A 0.000, B 0.000, C 0.000 }
gfCNCPoint3[12839] = {X 486.4706, Y 22.5736, Z -3.9499, A 0.000, B 0.000, C 0.000 }
gfCNCPoint3[12840] = {X 487.6448, Y 22.5560, Z -4.2646, A 0.000, B 0.000, C 0.000 }
gfCNCPoint3[12841] = {X 489.1454, Y 22.5560, Z -4.6667, A 0.000, B 0.000, C 0.000 }
gfCNCPoint3[12842] = {X 493.3690, Y 22.5560, Z -4.6667, A 0.000, B 0.000, C 0.000 }
gfCNCPoint3[12843] = {X 493.3690, Y 19.7819, Z -4.6667, A 0.000, B 0.000, C 0.000 }
gfCNCPoint3[12844] = {X 487.6645, Y 19.7811, Z -4.6667, A 0.000, B 0.000, C 0.000 }
gfCNCPoint3[12845] = {X 486.9699, Y 19.7858, Z -4.6667, A 0.000, B 0.000, C 0.000 }
gfCNCPoint3[12846] = {X 485.8746, Y 19.8570, Z -4.6667, A 0.000, B 0.000, C 0.000 }
gfCNCPoint3[12847] = {X 484.7986, Y 20.0737, Z -4.6667, A 0.000, B 0.000, C 0.000 }
gfCNCPoint3[12848] = {X 484.6683, Y 20.1467, Z -4.6667, A 0.000, B 0.000, C 0.000 }
gfCNCPoint3[12849] = {X 484.5876, Y 20.2724, Z -4.6667, A 0.000, B 0.000, C 0.000 }
gfCNCPoint3[12850] = {X 484.4293, Y 20.9578, Z -4.6667, A 0.000, B 0.000, C 0.000 }
gfCNCPoint3[12851] = {X 484.4088, Y 21.6609, Z -4.6667, A 0.000, B 0.000, C 0.000 }
gfCNCPoint3[12852] = {X 484.5268, Y 22.3544, Z -4.6667, A 0.000, B 0.000, C 0.000 }
gfCNCPoint3[12853] = {X 484.7284, Y 22.4071, Z -4.6667, A 0.000, B 0.000, C 0.000 }
gfCNCPoint3[12854] = {X 484.9348, Y 22.4355, Z -4.6667, A 0.000, B 0.000, C 0.000 }
gfCNCPoint3[12855] = {X 486.2880, Y 22.5362, Z -4.6667, A 0.000, B 0.000, C 0.000 }
gfCNCPoint3[12856] = {X 487.6448, Y 22.5560, Z -4.6667, A 0.000, B 0.000, C 0.000 }
gfCNCPoint3[12857] = {X 489.1454, Y 22.5560, Z -4.6667, A 0.000, B 0.000, C 0.000 }
gfCNCPoint3[12858] = {X 485.1607, Y 22.2874, Z -4.6667, A 0.000, B 0.000, C 0.000 }
gfCNCPoint3[12859] = {X 489.1454, Y 22.6360, Z -4.6667, A 0.000, B 0.000, C 0.000 }
gfCNCPoint3[12860] = {X 493.4490, Y 22.6360, Z -4.6667, A 0.000, B 0.000, C 0.000 }
gfCNCPoint3[12861] = {X 493.4490, Y 19.7019, Z -4.6667, A 0.000, B 0.000, C 0.000 }
gfCNCPoint3[12862] = {X 487.6642, Y 19.7011, Z -4.6667, A 0.000, B 0.000, C 0.000 }
gfCNCPoint3[12863] = {X 486.9714, Y 19.7058, Z -4.6667, A 0.000, B 0.000, C 0.000 }
gfCNCPoint3[12864] = {X 485.8648, Y 19.7776, Z -4.6667, A 0.000, B 0.000, C 0.000 }
gfCNCPoint3[12865] = {X 484.7776, Y 19.9965, Z -4.6667, A 0.000, B 0.000, C 0.000 }
gfCNCPoint3[12866] = {X 484.6135, Y 20.0884, Z -4.6667, A 0.000, B 0.000, C 0.000 }
gfCNCPoint3[12867] = {X 484.5118, Y 20.2468, Z -4.6667, A 0.000, B 0.000, C 0.000 }
gfCNCPoint3[12868] = {X 484.3482, Y 20.9617, Z -4.6667, A 0.000, B 0.000, C 0.000 }
gfCNCPoint3[12869] = {X 484.3311, Y 21.6949, Z -4.6667, A 0.000, B 0.000, C 0.000 }
gfCNCPoint3[12870] = {X 484.4612, Y 22.4167, Z -4.6667, A 0.000, B 0.000, C 0.000 }
gfCNCPoint3[12871] = {X 484.6889, Y 22.4806, Z -4.6667, A 0.000, B 0.000, C 0.000 }
gfCNCPoint3[12872] = {X 484.9229, Y 22.5147, Z -4.6667, A 0.000, B 0.000, C 0.000 }
gfCNCPoint3[12873] = {X 486.2809, Y 22.6160, Z -4.6667, A 0.000, B 0.000, C 0.000 }
gfCNCPoint3[12874] = {X 487.6424, Y 22.6360, Z -4.6667, A 0.000, B 0.000, C 0.000 }
gfCNCPoint3[12875] = {X 489.1454, Y 22.6360, Z -4.6667, A 0.000, B 0.000, C 0.000 }
gfCNCPoint3[12876] = {X 493.1302, Y 22.2874, Z -4.6667, A 0.000, B 0.000, C 0.000 }
gfCNCPoint3[12877] = {X 485.1607, Y 22.3674, Z -4.6667, A 0.000, B 0.000, C 0.000 }
gfCNCPoint3[12878] = {X 489.1454, Y 22.7160, Z -4.6667, A 0.000, B 0.000, C 0.000 }
gfCNCPoint3[12879] = {X 493.5290, Y 22.7160, Z -4.6667, A 0.000, B 0.000, C 0.000 }
gfCNCPoint3[12880] = {X 493.5290, Y 19.6219, Z -4.6667, A 0.000, B 0.000, C 0.000 }
gfCNCPoint3[12881] = {X 487.6640, Y 19.6211, Z -4.6667, A 0.000, B 0.000, C 0.000 }
gfCNCPoint3[12882] = {X 486.9712, Y 19.6258, Z -4.6667, A 0.000, B 0.000, C 0.000 }
gfCNCPoint3[12883] = {X 485.8541, Y 19.6983, Z -4.6667, A 0.000, B 0.000, C 0.000 }
gfCNCPoint3[12884] = {X 484.7566, Y 19.9193, Z -4.6667, A 0.000, B 0.000, C 0.000 }
gfCNCPoint3[12885] = {X 484.5586, Y 20.0302, Z -4.6667, A 0.000, B 0.000, C 0.000 }
gfCNCPoint3[12886] = {X 484.4360, Y 20.2212, Z -4.6667, A 0.000, B 0.000, C 0.000 }
gfCNCPoint3[12887] = {X 484.2672, Y 20.9653, Z -4.6667, A 0.000, B 0.000, C 0.000 }
gfCNCPoint3[12888] = {X 484.2536, Y 21.7283, Z -4.6667, A 0.000, B 0.000, C 0.000 }
gfCNCPoint3[12889] = {X 484.3958, Y 22.4780, Z -4.6667, A 0.000, B 0.000, C 0.000 }
gfCNCPoint3[12890] = {X 484.6516, Y 22.5543, Z -4.6667, A 0.000, B 0.000, C 0.000 }
gfCNCPoint3[12891] = {X 484.9155, Y 22.5944, Z -4.6667, A 0.000, B 0.000, C 0.000 }
gfCNCPoint3[12892] = {X 486.2774, Y 22.6959, Z -4.6667, A 0.000, B 0.000, C 0.000 }
gfCNCPoint3[12893] = {X 487.6430, Y 22.7160, Z -4.6667, A 0.000, B 0.000, C 0.000 }
gfCNCPoint3[12894] = {X 489.1454, Y 22.7160, Z -4.6667, A 0.000, B 0.000, C 0.000 }
gfCNCPoint3[12895] = {X 493.1302, Y 22.3674, Z -4.6667, A 0.000, B 0.000, C 0.000 }
gfCNCPoint3[12896] = {X 485.1607, Y 22.4474, Z -4.6667, A 0.000, B 0.000, C 0.000 }
gfCNCPoint3[12897] = {X 489.1454, Y 22.7960, Z -4.6667, A 0.000, B 0.000, C 0.000 }
gfCNCPoint3[12898] = {X 493.6090, Y 22.7960, Z -4.6667, A 0.000, B 0.000, C 0.000 }
gfCNCPoint3[12899] = {X 493.6090, Y 19.5419, Z -4.6667, A 0.000, B 0.000, C 0.000 }
gfCNCPoint3[12900] = {X 487.6637, Y 19.5411, Z -4.6667, A 0.000, B 0.000, C 0.000 }
gfCNCPoint3[12901] = {X 486.9711, Y 19.5458, Z -4.6667, A 0.000, B 0.000, C 0.000 }
gfCNCPoint3[12902] = {X 485.8434, Y 19.6190, Z -4.6667, A 0.000, B 0.000, C 0.000 }
gfCNCPoint3[12903] = {X 484.7356, Y 19.8421, Z -4.6667, A 0.000, B 0.000, C 0.000 }
gfCNCPoint3[12904] = {X 484.5038, Y 19.9719, Z -4.6667, A 0.000, B 0.000, C 0.000 }
gfCNCPoint3[12905] = {X 484.3602, Y 20.1955, Z -4.6667, A 0.000, B 0.000, C 0.000 }
gfCNCPoint3[12906] = {X 484.1862, Y 20.9687, Z -4.6667, A 0.000, B 0.000, C 0.000 }
gfCNCPoint3[12907] = {X 484.1762, Y 21.7612, Z -4.6667, A 0.000, B 0.000, C 0.000 }
gfCNCPoint3[12908] = {X 484.3306, Y 22.5386, Z -4.6667, A 0.000, B 0.000, C 0.000 }
gfCNCPoint3[12909] = {X 484.6143, Y 22.6278, Z -4.6667, A 0.000, B 0.000, C 0.000 }
gfCNCPoint3[12910] = {X 484.9081, Y 22.6740, Z -4.6667, A 0.000, B 0.000, C 0.000 }
gfCNCPoint3[12911] = {X 486.2740, Y 22.7758, Z -4.6667, A 0.000, B 0.000, C 0.000 }
gfCNCPoint3[12912] = {X 487.6436, Y 22.7960, Z -4.6667, A 0.000, B 0.000, C 0.000 }
gfCNCPoint3[12913] = {X 489.1454, Y 22.7960, Z -4.6667, A 0.000, B 0.000, C 0.000 }
gfCNCPoint3[12914] = {X 493.1302, Y 22.4474, Z -4.6667, A 0.000, B 0.000, C 0.000 }
gfCNCPoint3[12915] = {X 485.1607, Y 22.5274, Z -4.6667, A 0.000, B 0.000, C 0.000 }
gfCNCPoint3[12916] = {X 489.1454, Y 22.8760, Z -4.6667, A 0.000, B 0.000, C 0.000 }
gfCNCPoint3[12917] = {X 493.6890, Y 22.8760, Z -4.6667, A 0.000, B 0.000, C 0.000 }
gfCNCPoint3[12918] = {X 493.6890, Y 19.4619, Z -4.6667, A 0.000, B 0.000, C 0.000 }
gfCNCPoint3[12919] = {X 487.6634, Y 19.4611, Z -4.6667, A 0.000, B 0.000, C 0.000 }
gfCNCPoint3[12920] = {X 486.9709, Y 19.4658, Z -4.6667, A 0.000, B 0.000, C 0.000 }
gfCNCPoint3[12921] = {X 485.8327, Y 19.5397, Z -4.6667, A 0.000, B 0.000, C 0.000 }
gfCNCPoint3[12922] = {X 484.7146, Y 19.7649, Z -4.6667, A 0.000, B 0.000, C 0.000 }
gfCNCPoint3[12923] = {X 484.4489, Y 19.9137, Z -4.6667, A 0.000, B 0.000, C 0.000 }
gfCNCPoint3[12924] = {X 484.2845, Y 20.1699, Z -4.6667, A 0.000, B 0.000, C 0.000 }
gfCNCPoint3[12925] = {X 484.1053, Y 20.9719, Z -4.6667, A 0.000, B 0.000, C 0.000 }
gfCNCPoint3[12926] = {X 484.0989, Y 21.7937, Z -4.6667, A 0.000, B 0.000, C 0.000 }
gfCNCPoint3[12927] = {X 484.2656, Y 22.5984, Z -4.6667, A 0.000, B 0.000, C 0.000 }
gfCNCPoint3[12928] = {X 484.5770, Y 22.7011, Z -4.6667, A 0.000, B 0.000, C 0.000 }
gfCNCPoint3[12929] = {X 484.9007, Y 22.7537, Z -4.6667, A 0.000, B 0.000, C 0.000 }
gfCNCPoint3[12930] = {X 486.2706, Y 22.8558, Z -4.6667, A 0.000, B 0.000, C 0.000 }
gfCNCPoint3[12931] = {X 487.6442, Y 22.8760, Z -4.6667, A 0.000, B 0.000, C 0.000 }
gfCNCPoint3[12932] = {X 489.1454, Y 22.8760, Z -4.6667, A 0.000, B 0.000, C 0.000 }
gfCNCPoint3[12933] = {X 493.1302, Y 22.5274, Z -4.6667, A 0.000, B 0.000, C 0.000 }
gfCNCPoint3[12934] = {X 485.1607, Y 22.6074, Z -4.6667, A 0.000, B 0.000, C 0.000 }
gfCNCPoint3[12935] = {X 489.1454, Y 22.9560, Z -4.6667, A 0.000, B 0.000, C 0.000 }
gfCNCPoint3[12936] = {X 493.7690, Y 22.9560, Z -4.6667, A 0.000, B 0.000, C 0.000 }
gfCNCPoint3[12937] = {X 493.7695, Y 19.3819, Z -4.6667, A 0.000, B 0.000, C 0.000 }
gfCNCPoint3[12938] = {X 487.6632, Y 19.3811, Z -4.6667, A 0.000, B 0.000, C 0.000 }
gfCNCPoint3[12939] = {X 486.9707, Y 19.3858, Z -4.6667, A 0.000, B 0.000, C 0.000 }
gfCNCPoint3[12940] = {X 485.8220, Y 19.4605, Z -4.6667, A 0.000, B 0.000, C 0.000 }
gfCNCPoint3[12941] = {X 484.6936, Y 19.6877, Z -4.6667, A 0.000, B 0.000, C 0.000 }
gfCNCPoint3[12942] = {X 484.3941, Y 19.8554, Z -4.6667, A 0.000, B 0.000, C 0.000 }
gfCNCPoint3[12943] = {X 484.2087, Y 20.1443, Z -4.6667, A 0.000, B 0.000, C 0.000 }
gfCNCPoint3[12944] = {X 484.0244, Y 20.9750, Z -4.6667, A 0.000, B 0.000, C 0.000 }
gfCNCPoint3[12945] = {X 484.0217, Y 21.8258, Z -4.6667, A 0.000, B 0.000, C 0.000 }
gfCNCPoint3[12946] = {X 484.2007, Y 22.6576, Z -4.6667, A 0.000, B 0.000, C 0.000 }
gfCNCPoint3[12947] = {X 484.5397, Y 22.7743, Z -4.6667, A 0.000, B 0.000, C 0.000 }
gfCNCPoint3[12948] = {X 484.8932, Y 22.8334, Z -4.6667, A 0.000, B 0.000, C 0.000 }
gfCNCPoint3[12949] = {X 486.2672, Y 22.9357, Z -4.6667, A 0.000, B 0.000, C 0.000 }
gfCNCPoint3[12950] = {X 487.6448, Y 22.9560, Z -4.6667, A 0.000, B 0.000, C 0.000 }
gfCNCPoint3[12951] = {X 489.1454, Y 22.9560, Z -4.6667, A 0.000, B 0.000, C 0.000 }
gfCNCPoint3[12952] = {X 493.1302, Y 22.6074, Z -4.6667, A 0.000, B 0.000, C 0.000 }
gfCNCPoint3[12953] = {X 493.1302, Y 22.6074, Z -1.6667, A 0.000, B 0.000, C 0.000 }
gfCNCPoint3[12954] = {X 493.1302, Y 22.6074, Z 11.0000, A 0.000, B 0.000, C 0.000 }
gfCNCPoint3[12955] = {X 448.7135, Y 19.7819, Z 11.0000, A 0.000, B 0.000, C 0.000 }
gfCNCPoint3[12956] = {X 448.7135, Y 19.7819, Z -0.8333, A 0.000, B 0.000, C 0.000 }
gfCNCPoint3[12957] = {X 444.0413, Y 19.7818, Z -2.0852, A 0.000, B 0.000, C 0.000 }
gfCNCPoint3[12958] = {X 443.3488, Y 19.7980, Z -2.2709, A 0.000, B 0.000, C 0.000 }
gfCNCPoint3[12959] = {X 442.7487, Y 19.8048, Z -2.4317, A 0.000, B 0.000, C 0.000 }
gfCNCPoint3[12960] = {X 442.0370, Y 19.9280, Z -2.6252, A 0.000, B 0.000, C 0.000 }
gfCNCPoint3[12961] = {X 441.3665, Y 20.1587, Z -2.8152, A 0.000, B 0.000, C 0.000 }
gfCNCPoint3[12962] = {X 441.1887, Y 20.7183, Z -2.9725, A 0.000, B 0.000, C 0.000 }
gfCNCPoint3[12963] = {X 441.1550, Y 21.8882, Z -3.2861, A 0.000, B 0.000, C 0.000 }
gfCNCPoint3[12964] = {X 441.2734, Y 22.3515, Z -3.4143, A 0.000, B 0.000, C 0.000 }
gfCNCPoint3[12965] = {X 441.5028, Y 22.4265, Z -3.4789, A 0.000, B 0.000, C 0.000 }
gfCNCPoint3[12966] = {X 442.9982, Y 22.5626, Z -3.8813, A 0.000, B 0.000, C 0.000 }
gfCNCPoint3[12967] = {X 443.1303, Y 22.5680, Z -3.9167, A 0.000, B 0.000, C 0.000 }
gfCNCPoint3[12968] = {X 444.3942, Y 22.5560, Z -4.2554, A 0.000, B 0.000, C 0.000 }
gfCNCPoint3[12969] = {X 445.9292, Y 22.5560, Z -4.6667, A 0.000, B 0.000, C 0.000 }
gfCNCPoint3[12970] = {X 450.1184, Y 22.5560, Z -4.6667, A 0.000, B 0.000, C 0.000 }
gfCNCPoint3[12971] = {X 450.1184, Y 19.7819, Z -4.6667, A 0.000, B 0.000, C 0.000 }
gfCNCPoint3[12972] = {X 444.0413, Y 19.7818, Z -4.6667, A 0.000, B 0.000, C 0.000 }
gfCNCPoint3[12973] = {X 443.3488, Y 19.7980, Z -4.6667, A 0.000, B 0.000, C 0.000 }
gfCNCPoint3[12974] = {X 442.3961, Y 19.8853, Z -4.6667, A 0.000, B 0.000, C 0.000 }
gfCNCPoint3[12975] = {X 441.4696, Y 20.1232, Z -4.6667, A 0.000, B 0.000, C 0.000 }
gfCNCPoint3[12976] = {X 441.3850, Y 20.1768, Z -4.6667, A 0.000, B 0.000, C 0.000 }
gfCNCPoint3[12977] = {X 441.3335, Y 20.2626, Z -4.6667, A 0.000, B 0.000, C 0.000 }
gfCNCPoint3[12978] = {X 441.1834, Y 20.9511, Z -4.6667, A 0.000, B 0.000, C 0.000 }
gfCNCPoint3[12979] = {X 441.1631, Y 21.6555, Z -4.6667, A 0.000, B 0.000, C 0.000 }
gfCNCPoint3[12980] = {X 441.2734, Y 22.3515, Z -4.6667, A 0.000, B 0.000, C 0.000 }
gfCNCPoint3[12981] = {X 441.5055, Y 22.4132, Z -4.6667, A 0.000, B 0.000, C 0.000 }
gfCNCPoint3[12982] = {X 441.7432, Y 22.4484, Z -4.6667, A 0.000, B 0.000, C 0.000 }
gfCNCPoint3[12983] = {X 443.0673, Y 22.5355, Z -4.6667, A 0.000, B 0.000, C 0.000 }
gfCNCPoint3[12984] = {X 444.3942, Y 22.5560, Z -4.6667, A 0.000, B 0.000, C 0.000 }
gfCNCPoint3[12985] = {X 445.9292, Y 22.5560, Z -4.6667, A 0.000, B 0.000, C 0.000 }
gfCNCPoint3[12986] = {X 441.9444, Y 22.2874, Z -4.6667, A 0.000, B 0.000, C 0.000 }
gfCNCPoint3[12987] = {X 445.9292, Y 22.6360, Z -4.6667, A 0.000, B 0.000, C 0.000 }
gfCNCPoint3[12988] = {X 450.1984, Y 22.6360, Z -4.6667, A 0.000, B 0.000, C 0.000 }
gfCNCPoint3[12989] = {X 450.1984, Y 19.7019, Z -4.6667, A 0.000, B 0.000, C 0.000 }
gfCNCPoint3[12990] = {X 444.0404, Y 19.7018, Z -4.6667, A 0.000, B 0.000, C 0.000 }
gfCNCPoint3[12991] = {X 443.3497, Y 19.7179, Z -4.6667, A 0.000, B 0.000, C 0.000 }
gfCNCPoint3[12992] = {X 442.3834, Y 19.8063, Z -4.6667, A 0.000, B 0.000, C 0.000 }
gfCNCPoint3[12993] = {X 441.4436, Y 20.0476, Z -4.6667, A 0.000, B 0.000, C 0.000 }
gfCNCPoint3[12994] = {X 441.3278, Y 20.1209, Z -4.6667, A 0.000, B 0.000, C 0.000 }
gfCNCPoint3[12995] = {X 441.2573, Y 20.2383, Z -4.6667, A 0.000, B 0.000, C 0.000 }
gfCNCPoint3[12996] = {X 441.1022, Y 20.9558, Z -4.6667, A 0.000, B 0.000, C 0.000 }
gfCNCPoint3[12997] = {X 441.0852, Y 21.6896, Z -4.6667, A 0.000, B 0.000, C 0.000 }
gfCNCPoint3[12998] = {X 441.2069, Y 22.4135, Z -4.6667, A 0.000, B 0.000, C 0.000 }
gfCNCPoint3[12999] = {X 441.4679, Y 22.4870, Z -4.6667, A 0.000, B 0.000, C 0.000 }
gfCNCPoint3[13000] = {X 441.7359, Y 22.5281, Z -4.6667, A 0.000, B 0.000, C 0.000 }
gfCNCPoint3[13001] = {X 443.0630, Y 22.6154, Z -4.6667, A 0.000, B 0.000, C 0.000 }
gfCNCPoint3[13002] = {X 444.3927, Y 22.6360, Z -4.6667, A 0.000, B 0.000, C 0.000 }
gfCNCPoint3[13003] = {X 445.9292, Y 22.6360, Z -4.6667, A 0.000, B 0.000, C 0.000 }
gfCNCPoint3[13004] = {X 449.9139, Y 22.2874, Z -4.6667, A 0.000, B 0.000, C 0.000 }
gfCNCPoint3[13005] = {X 441.9444, Y 22.3674, Z -4.6667, A 0.000, B 0.000, C 0.000 }
gfCNCPoint3[13006] = {X 445.9292, Y 22.7160, Z -4.6667, A 0.000, B 0.000, C 0.000 }
gfCNCPoint3[13007] = {X 450.2784, Y 22.7160, Z -4.6667, A 0.000, B 0.000, C 0.000 }
gfCNCPoint3[13008] = {X 450.2784, Y 19.6219, Z -4.6667, A 0.000, B 0.000, C 0.000 }
gfCNCPoint3[13009] = {X 444.0395, Y 19.6218, Z -4.6667, A 0.000, B 0.000, C 0.000 }
gfCNCPoint3[13010] = {X 443.3484, Y 19.6380, Z -4.6667, A 0.000, B 0.000, C 0.000 }
gfCNCPoint3[13011] = {X 442.3695, Y 19.7275, Z -4.6667, A 0.000, B 0.000, C 0.000 }
gfCNCPoint3[13012] = {X 441.4175, Y 19.9719, Z -4.6667, A 0.000, B 0.000, C 0.000 }
gfCNCPoint3[13013] = {X 441.2706, Y 20.0650, Z -4.6667, A 0.000, B 0.000, C 0.000 }
gfCNCPoint3[13014] = {X 441.1810, Y 20.2141, Z -4.6667, A 0.000, B 0.000, C 0.000 }
gfCNCPoint3[13015] = {X 441.0212, Y 20.9603, Z -4.6667, A 0.000, B 0.000, C 0.000 }
gfCNCPoint3[13016] = {X 441.0076, Y 21.7233, Z -4.6667, A 0.000, B 0.000, C 0.000 }
gfCNCPoint3[13017] = {X 441.1407, Y 22.4747, Z -4.6667, A 0.000, B 0.000, C 0.000 }
gfCNCPoint3[13018] = {X 441.4303, Y 22.5606, Z -4.6667, A 0.000, B 0.000, C 0.000 }
gfCNCPoint3[13019] = {X 441.7287, Y 22.6077, Z -4.6667, A 0.000, B 0.000, C 0.000 }
gfCNCPoint3[13020] = {X 443.0595, Y 22.6953, Z -4.6667, A 0.000, B 0.000, C 0.000 }
gfCNCPoint3[13021] = {X 444.3931, Y 22.7160, Z -4.6667, A 0.000, B 0.000, C 0.000 }
gfCNCPoint3[13022] = {X 445.9292, Y 22.7160, Z -4.6667, A 0.000, B 0.000, C 0.000 }
gfCNCPoint3[13023] = {X 449.9139, Y 22.3674, Z -4.6667, A 0.000, B 0.000, C 0.000 }
gfCNCPoint3[13024] = {X 441.9444, Y 22.4474, Z -4.6667, A 0.000, B 0.000, C 0.000 }
gfCNCPoint3[13025] = {X 445.9292, Y 22.7960, Z -4.6667, A 0.000, B 0.000, C 0.000 }
gfCNCPoint3[13026] = {X 450.3584, Y 22.7960, Z -4.6667, A 0.000, B 0.000, C 0.000 }
gfCNCPoint3[13027] = {X 450.3584, Y 19.5419, Z -4.6667, A 0.000, B 0.000, C 0.000 }
gfCNCPoint3[13028] = {X 444.0385, Y 19.5418, Z -4.6667, A 0.000, B 0.000, C 0.000 }
gfCNCPoint3[13029] = {X 443.3470, Y 19.5580, Z -4.6667, A 0.000, B 0.000, C 0.000 }
gfCNCPoint3[13030] = {X 442.3557, Y 19.6487, Z -4.6667, A 0.000, B 0.000, C 0.000 }
gfCNCPoint3[13031] = {X 441.3915, Y 19.8963, Z -4.6667, A 0.000, B 0.000, C 0.000 }
gfCNCPoint3[13032] = {X 441.2133, Y 20.0091, Z -4.6667, A 0.000, B 0.000, C 0.000 }
gfCNCPoint3[13033] = {X 441.1048, Y 20.1899, Z -4.6667, A 0.000, B 0.000, C 0.000 }
gfCNCPoint3[13034] = {X 440.9402, Y 20.9646, Z -4.6667, A 0.000, B 0.000, C 0.000 }
gfCNCPoint3[13035] = {X 440.9300, Y 21.7565, Z -4.6667, A 0.000, B 0.000, C 0.000 }
gfCNCPoint3[13036] = {X 441.0747, Y 22.5352, Z -4.6667, A 0.000, B 0.000, C 0.000 }
gfCNCPoint3[13037] = {X 441.3927, Y 22.6340, Z -4.6667, A 0.000, B 0.000, C 0.000 }
gfCNCPoint3[13038] = {X 441.7214, Y 22.6874, Z -4.6667, A 0.000, B 0.000, C 0.000 }
gfCNCPoint3[13039] = {X 443.0561, Y 22.7752, Z -4.6667, A 0.000, B 0.000, C 0.000 }
gfCNCPoint3[13040] = {X 444.3935, Y 22.7960, Z -4.6667, A 0.000, B 0.000, C 0.000 }
gfCNCPoint3[13041] = {X 445.9292, Y 22.7960, Z -4.6667, A 0.000, B 0.000, C 0.000 }
gfCNCPoint3[13042] = {X 449.9139, Y 22.4474, Z -4.6667, A 0.000, B 0.000, C 0.000 }
gfCNCPoint3[13043] = {X 441.9444, Y 22.5274, Z -4.6667, A 0.000, B 0.000, C 0.000 }
gfCNCPoint3[13044] = {X 445.9292, Y 22.8760, Z -4.6667, A 0.000, B 0.000, C 0.000 }
gfCNCPoint3[13045] = {X 450.4384, Y 22.8760, Z -4.6667, A 0.000, B 0.000, C 0.000 }
gfCNCPoint3[13046] = {X 450.4384, Y 19.4619, Z -4.6667, A 0.000, B 0.000, C 0.000 }
gfCNCPoint3[13047] = {X 444.0376, Y 19.4618, Z -4.6667, A 0.000, B 0.000, C 0.000 }
gfCNCPoint3[13048] = {X 443.3456, Y 19.4780, Z -4.6667, A 0.000, B 0.000, C 0.000 }
gfCNCPoint3[13049] = {X 442.3418, Y 19.5699, Z -4.6667, A 0.000, B 0.000, C 0.000 }
gfCNCPoint3[13050] = {X 441.3655, Y 19.8206, Z -4.6667, A 0.000, B 0.000, C 0.000 }
gfCNCPoint3[13051] = {X 441.1561, Y 19.9532, Z -4.6667, A 0.000, B 0.000, C 0.000 }
gfCNCPoint3[13052] = {X 441.0286, Y 20.1657, Z -4.6667, A 0.000, B 0.000, C 0.000 }
gfCNCPoint3[13053] = {X 440.8592, Y 20.9687, Z -4.6667, A 0.000, B 0.000, C 0.000 }
gfCNCPoint3[13054] = {X 440.8526, Y 21.7894, Z -4.6667, A 0.000, B 0.000, C 0.000 }
gfCNCPoint3[13055] = {X 441.0090, Y 22.5951, Z -4.6667, A 0.000, B 0.000, C 0.000 }
gfCNCPoint3[13056] = {X 441.3552, Y 22.7073, Z -4.6667, A 0.000, B 0.000, C 0.000 }
gfCNCPoint3[13057] = {X 441.7142, Y 22.7671, Z -4.6667, A 0.000, B 0.000, C 0.000 }
gfCNCPoint3[13058] = {X 443.0526, Y 22.8551, Z -4.6667, A 0.000, B 0.000, C 0.000 }
gfCNCPoint3[13059] = {X 444.3939, Y 22.8760, Z -4.6667, A 0.000, B 0.000, C 0.000 }
gfCNCPoint3[13060] = {X 445.9292, Y 22.8760, Z -4.6667, A 0.000, B 0.000, C 0.000 }
gfCNCPoint3[13061] = {X 449.9139, Y 22.5274, Z -4.6667, A 0.000, B 0.000, C 0.000 }
gfCNCPoint3[13062] = {X 441.9444, Y 22.6074, Z -4.6667, A 0.000, B 0.000, C 0.000 }
gfCNCPoint3[13063] = {X 445.9292, Y 22.9560, Z -4.6667, A 0.000, B 0.000, C 0.000 }
gfCNCPoint3[13064] = {X 450.5184, Y 22.9560, Z -4.6667, A 0.000, B 0.000, C 0.000 }
gfCNCPoint3[13065] = {X 450.5189, Y 19.3819, Z -4.6667, A 0.000, B 0.000, C 0.000 }
gfCNCPoint3[13066] = {X 444.0367, Y 19.3818, Z -4.6667, A 0.000, B 0.000, C 0.000 }
gfCNCPoint3[13067] = {X 443.3442, Y 19.3980, Z -4.6667, A 0.000, B 0.000, C 0.000 }
gfCNCPoint3[13068] = {X 442.3279, Y 19.4911, Z -4.6667, A 0.000, B 0.000, C 0.000 }
gfCNCPoint3[13069] = {X 441.3395, Y 19.7450, Z -4.6667, A 0.000, B 0.000, C 0.000 }
gfCNCPoint3[13070] = {X 441.0989, Y 19.8973, Z -4.6667, A 0.000, B 0.000, C 0.000 }
gfCNCPoint3[13071] = {X 440.9523, Y 20.1414, Z -4.6667, A 0.000, B 0.000, C 0.000 }
gfCNCPoint3[13072] = {X 440.7784, Y 20.9727, Z -4.6667, A 0.000, B 0.000, C 0.000 }
gfCNCPoint3[13073] = {X 440.7754, Y 21.8219, Z -4.6667, A 0.000, B 0.000, C 0.000 }
gfCNCPoint3[13074] = {X 440.9434, Y 22.6544, Z -4.6667, A 0.000, B 0.000, C 0.000 }
gfCNCPoint3[13075] = {X 441.3176, Y 22.7804, Z -4.6667, A 0.000, B 0.000, C 0.000 }
gfCNCPoint3[13076] = {X 441.7069, Y 22.8468, Z -4.6667, A 0.000, B 0.000, C 0.000 }
gfCNCPoint3[13077] = {X 443.0492, Y 22.9351, Z -4.6667, A 0.000, B 0.000, C 0.000 }
gfCNCPoint3[13078] = {X 444.3942, Y 22.9560, Z -4.6667, A 0.000, B 0.000, C 0.000 }
gfCNCPoint3[13079] = {X 445.9292, Y 22.9560, Z -4.6667, A 0.000, B 0.000, C 0.000 }
gfCNCPoint3[13080] = {X 449.9139, Y 22.6074, Z -4.6667, A 0.000, B 0.000, C 0.000 }
gfCNCPoint3[13081] = {X 449.9139, Y 22.6074, Z -1.6667, A 0.000, B 0.000, C 0.000 }
gfCNCPoint3[13082] = {X 449.9139, Y 22.6074, Z 11.0000, A 0.000, B 0.000, C 0.000 }
gfCNCPoint3[13083] = {X 507.6815, Y 107.6950, Z 11.0000, A 0.000, B 0.000, C 0.000 }
gfCNCPoint3[13084] = {X 507.6815, Y 107.6950, Z -1.6667, A 0.000, B 0.000, C 0.000 }
gfCNCPoint3[13085] = {X 507.6815, Y 107.6950, Z -4.6667, A 0.000, B 0.000, C 0.000 }
gfCNCPoint3[13086] = {X 507.6815, Y 71.2950, Z -4.6667, A 0.000, B 0.000, C 0.000 }
gfCNCPoint3[13087] = {X 509.5502, Y 71.2950, Z -4.6667, A 0.000, B 0.000, C 0.000 }
gfCNCPoint3[13088] = {X 509.0279, Y 71.0691, Z -4.6667, A 0.000, B 0.000, C 0.000 }
gfCNCPoint3[13089] = {X 508.5105, Y 70.8320, Z -4.6667, A 0.000, B 0.000, C 0.000 }
gfCNCPoint3[13090] = {X 507.1677, Y 71.0984, Z -4.6667, A 0.000, B 0.000, C 0.000 }
gfCNCPoint3[13091] = {X 505.8129, Y 71.2950, Z -4.6667, A 0.000, B 0.000, C 0.000 }
gfCNCPoint3[13092] = {X 507.6815, Y 71.2950, Z -4.6667, A 0.000, B 0.000, C 0.000 }
gfCNCPoint3[13093] = {X 507.6815, Y 73.6950, Z -4.6667, A 0.000, B 0.000, C 0.000 }
gfCNCPoint3[13094] = {X 551.2534, Y 73.6950, Z -4.6667, A 0.000, B 0.000, C 0.000 }
gfCNCPoint3[13095] = {X 549.1238, Y 72.7706, Z -4.6667, A 0.000, B 0.000, C 0.000 }
gfCNCPoint3[13096] = {X 547.0699, Y 71.6883, Z -4.6667, A 0.000, B 0.000, C 0.000 }
gfCNCPoint3[13097] = {X 545.1033, Y 70.4544, Z -4.6667, A 0.000, B 0.000, C 0.000 }
gfCNCPoint3[13098] = {X 543.2352, Y 69.0759, Z -4.6667, A 0.000, B 0.000, C 0.000 }
gfCNCPoint3[13099] = {X 529.7634, Y 69.0762, Z -4.6667, A 0.000, B 0.000, C 0.000 }
gfCNCPoint3[13100] = {X 527.5600, Y 69.8766, Z -4.6667, A 0.000, B 0.000, C 0.000 }
gfCNCPoint3[13101] = {X 525.2896, Y 70.4605, Z -4.6667, A 0.000, B 0.000, C 0.000 }
gfCNCPoint3[13102] = {X 522.9735, Y 70.8222, Z -4.6667, A 0.000, B 0.000, C 0.000 }
gfCNCPoint3[13103] = {X 520.6332, Y 70.9585, Z -4.6667, A 0.000, B 0.000, C 0.000 }
gfCNCPoint3[13104] = {X 519.7998, Y 70.9591, Z -4.6667, A 0.000, B 0.000, C 0.000 }
gfCNCPoint3[13105] = {X 517.4111, Y 70.8403, Z -4.6667, A 0.000, B 0.000, C 0.000 }
gfCNCPoint3[13106] = {X 515.0459, Y 70.4852, Z -4.6667, A 0.000, B 0.000, C 0.000 }
gfCNCPoint3[13107] = {X 512.7277, Y 69.8972, Z -4.6667, A 0.000, B 0.000, C 0.000 }
gfCNCPoint3[13108] = {X 510.4792, Y 69.0821, Z -4.6667, A 0.000, B 0.000, C 0.000 }
gfCNCPoint3[13109] = {X 509.6265, Y 68.7046, Z -4.6667, A 0.000, B 0.000, C 0.000 }
gfCNCPoint3[13110] = {X 508.7892, Y 68.2944, Z -4.6667, A 0.000, B 0.000, C 0.000 }
gfCNCPoint3[13111] = {X 507.1701, Y 68.6593, Z -4.6667, A 0.000, B 0.000, C 0.000 }
gfCNCPoint3[13112] = {X 505.5297, Y 68.9118, Z -4.6667, A 0.000, B 0.000, C 0.000 }
gfCNCPoint3[13113] = {X 504.1116, Y 69.0379, Z -4.6667, A 0.000, B 0.000, C 0.000 }
gfCNCPoint3[13114] = {X 502.6885, Y 69.0800, Z -4.6667, A 0.000, B 0.000, C 0.000 }
gfCNCPoint3[13115] = {X 502.0391, Y 69.0800, Z -4.6667, A 0.000, B 0.000, C 0.000 }
gfCNCPoint3[13116] = {X 501.1775, Y 71.1322, Z -4.6667, A 0.000, B 0.000, C 0.000 }
gfCNCPoint3[13117] = {X 500.1604, Y 73.1119, Z -4.6667, A 0.000, B 0.000, C 0.000 }
gfCNCPoint3[13118] = {X 500.1604, Y 73.6950, Z -4.6667, A 0.000, B 0.000, C 0.000 }
gfCNCPoint3[13119] = {X 507.6815, Y 73.6950, Z -4.6667, A 0.000, B 0.000, C 0.000 }
gfCNCPoint3[13120] = {X 507.6815, Y 76.0950, Z -4.6667, A 0.000, B 0.000, C 0.000 }
gfCNCPoint3[13121] = {X 576.0966, Y 76.0950, Z -4.6667, A 0.000, B 0.000, C 0.000 }
gfCNCPoint3[13122] = {X 576.0966, Y 72.8901, Z -4.6667, A 0.000, B 0.000, C 0.000 }
gfCNCPoint3[13123] = {X 575.7178, Y 72.8147, Z -4.6667, A 0.000, B 0.000, C 0.000 }
gfCNCPoint3[13124] = {X 575.3401, Y 72.7341, Z -4.6667, A 0.000, B 0.000, C 0.000 }
gfCNCPoint3[13125] = {X 573.3201, Y 73.1034, Z -4.6667, A 0.000, B 0.000, C 0.000 }
gfCNCPoint3[13126] = {X 571.2786, Y 73.3258, Z -4.6667, A 0.000, B 0.000, C 0.000 }
gfCNCPoint3[13127] = {X 569.2264, Y 73.4000, Z -4.6667, A 0.000, B 0.000, C 0.000 }
gfCNCPoint3[13128] = {X 562.4443, Y 73.4000, Z -4.6667, A 0.000, B 0.000, C 0.000 }
gfCNCPoint3[13129] = {X 560.3341, Y 73.3215, Z -4.6667, A 0.000, B 0.000, C 0.000 }
gfCNCPoint3[13130] = {X 558.2356, Y 73.0864, Z -4.6667, A 0.000, B 0.000, C 0.000 }
gfCNCPoint3[13131] = {X 556.1604, Y 72.6961, Z -4.6667, A 0.000, B 0.000, C 0.000 }
gfCNCPoint3[13132] = {X 554.1199, Y 72.1526, Z -4.6667, A 0.000, B 0.000, C 0.000 }
gfCNCPoint3[13133] = {X 552.1255, Y 71.4591, Z -4.6667, A 0.000, B 0.000, C 0.000 }
gfCNCPoint3[13134] = {X 549.9762, Y 70.5168, Z -4.6667, A 0.000, B 0.000, C 0.000 }
gfCNCPoint3[13135] = {X 547.9121, Y 69.4003, Z -4.6667, A 0.000, B 0.000, C 0.000 }
gfCNCPoint3[13136] = {X 545.9472, Y 68.1172, Z -4.6667, A 0.000, B 0.000, C 0.000 }
gfCNCPoint3[13137] = {X 544.0950, Y 66.6763, Z -4.6667, A 0.000, B 0.000, C 0.000 }
gfCNCPoint3[13138] = {X 543.8500, Y 66.6775, Z -4.6667, A 0.000, B 0.000, C 0.000 }
gfCNCPoint3[13139] = {X 543.6050, Y 66.6759, Z -4.6667, A 0.000, B 0.000, C 0.000 }
gfCNCPoint3[13140] = {X 529.2677, Y 66.6762, Z -4.6667, A 0.000, B 0.000, C 0.000 }
gfCNCPoint3[13141] = {X 527.1868, Y 67.4769, Z -4.6667, A 0.000, B 0.000, C 0.000 }
gfCNCPoint3[13142] = {X 525.0351, Y 68.0612, Z -4.6667, A 0.000, B 0.000, C 0.000 }
gfCNCPoint3[13143] = {X 522.8350, Y 68.4230, Z -4.6667, A 0.000, B 0.000, C 0.000 }
gfCNCPoint3[13144] = {X 520.6095, Y 68.5586, Z -4.6667, A 0.000, B 0.000, C 0.000 }
gfCNCPoint3[13145] = {X 519.7998, Y 68.5591, Z -4.6667, A 0.000, B 0.000, C 0.000 }
gfCNCPoint3[13146] = {X 517.5593, Y 68.4430, Z -4.6667, A 0.000, B 0.000, C 0.000 }
gfCNCPoint3[13147] = {X 515.3429, Y 68.0961, Z -4.6667, A 0.000, B 0.000, C 0.000 }
gfCNCPoint3[13148] = {X 513.1742, Y 67.5219, Z -4.6667, A 0.000, B 0.000, C 0.000 }
gfCNCPoint3[13149] = {X 511.0764, Y 66.7267, Z -4.6667, A 0.000, B 0.000, C 0.000 }
gfCNCPoint3[13150] = {X 509.0720, Y 65.7189, Z -4.6667, A 0.000, B 0.000, C 0.000 }
gfCNCPoint3[13151] = {X 506.9797, Y 66.2511, Z -4.6667, A 0.000, B 0.000, C 0.000 }
gfCNCPoint3[13152] = {X 504.8448, Y 66.5725, Z -4.6667, A 0.000, B 0.000, C 0.000 }
gfCNCPoint3[13153] = {X 502.6885, Y 66.6800, Z -4.6667, A 0.000, B 0.000, C 0.000 }
gfCNCPoint3[13154] = {X 500.3217, Y 66.6800, Z -4.6667, A 0.000, B 0.000, C 0.000 }
gfCNCPoint3[13155] = {X 499.6231, Y 68.6754, Z -4.6667, A 0.000, B 0.000, C 0.000 }
gfCNCPoint3[13156] = {X 498.7675, Y 70.6087, Z -4.6667, A 0.000, B 0.000, C 0.000 }
gfCNCPoint3[13157] = {X 497.7604, Y 72.4676, Z -4.6667, A 0.000, B 0.000, C 0.000 }
gfCNCPoint3[13158] = {X 497.7604, Y 76.0950, Z -4.6667, A 0.000, B 0.000, C 0.000 }
gfCNCPoint3[13159] = {X 507.6815, Y 76.0950, Z -4.6667, A 0.000, B 0.000, C 0.000 }
gfCNCPoint3[13160] = {X 507.6815, Y 78.4950, Z -4.6667, A 0.000, B 0.000, C 0.000 }
gfCNCPoint3[13161] = {X 578.4966, Y 78.4950, Z -4.6667, A 0.000, B 0.000, C 0.000 }
gfCNCPoint3[13162] = {X 578.4966, Y 70.8313, Z -4.6667, A 0.000, B 0.000, C 0.000 }
gfCNCPoint3[13163] = {X 576.9097, Y 70.5998, Z -4.6667, A 0.000, B 0.000, C 0.000 }
gfCNCPoint3[13164] = {X 575.3401, Y 70.2710, Z -4.6667, A 0.000, B 0.000, C 0.000 }
gfCNCPoint3[13165] = {X 573.3236, Y 70.6751, Z -4.6667, A 0.000, B 0.000, C 0.000 }
gfCNCPoint3[13166] = {X 571.2815, Y 70.9187, Z -4.6667, A 0.000, B 0.000, C 0.000 }
gfCNCPoint3[13167] = {X 569.2264, Y 71.0000, Z -4.6667, A 0.000, B 0.000, C 0.000 }
gfCNCPoint3[13168] = {X 562.4443, Y 71.0000, Z -4.6667, A 0.000, B 0.000, C 0.000 }
gfCNCPoint3[13169] = {X 560.0513, Y 70.8896, Z -4.6667, A 0.000, B 0.000, C 0.000 }
gfCNCPoint3[13170] = {X 557.6785, Y 70.5595, Z -4.6667, A 0.000, B 0.000, C 0.000 }
gfCNCPoint3[13171] = {X 555.3463, Y 70.0124, Z -4.6667, A 0.000, B 0.000, C 0.000 }
gfCNCPoint3[13172] = {X 553.0742, Y 69.2529, Z -4.6667, A 0.000, B 0.000, C 0.000 }
gfCNCPoint3[13173] = {X 550.8818, Y 68.2875, Z -4.6667, A 0.000, B 0.000, C 0.000 }
gfCNCPoint3[13174] = {X 548.7875, Y 67.1244, Z -4.6667, A 0.000, B 0.000, C 0.000 }
gfCNCPoint3[13175] = {X 546.8091, Y 65.7736, Z -4.6667, A 0.000, B 0.000, C 0.000 }
gfCNCPoint3[13176] = {X 544.9635, Y 64.2463, Z -4.6667, A 0.000, B 0.000, C 0.000 }
gfCNCPoint3[13177] = {X 544.2919, Y 64.2728, Z -4.6667, A 0.000, B 0.000, C 0.000 }
gfCNCPoint3[13178] = {X 543.6199, Y 64.2759, Z -4.6667, A 0.000, B 0.000, C 0.000 }
gfCNCPoint3[13179] = {X 528.7426, Y 64.2763, Z -4.6667, A 0.000, B 0.000, C 0.000 }
gfCNCPoint3[13180] = {X 526.7923, Y 65.0770, Z -4.6667, A 0.000, B 0.000, C 0.000 }
gfCNCPoint3[13181] = {X 524.7668, Y 65.6618, Z -4.6667, A 0.000, B 0.000, C 0.000 }
gfCNCPoint3[13182] = {X 522.6898, Y 66.0238, Z -4.6667, A 0.000, B 0.000, C 0.000 }
gfCNCPoint3[13183] = {X 520.5858, Y 66.1587, Z -4.6667, A 0.000, B 0.000, C 0.000 }
gfCNCPoint3[13184] = {X 519.7998, Y 66.1591, Z -4.6667, A 0.000, B 0.000, C 0.000 }
gfCNCPoint3[13185] = {X 517.9641, Y 66.0715, Z -4.6667, A 0.000, B 0.000, C 0.000 }
gfCNCPoint3[13186] = {X 516.1450, Y 65.8096, Z -4.6667, A 0.000, B 0.000, C 0.000 }
gfCNCPoint3[13187] = {X 514.3592, Y 65.3756, Z -4.6667, A 0.000, B 0.000, C 0.000 }
gfCNCPoint3[13188] = {X 512.6228, Y 64.7735, Z -4.6667, A 0.000, B 0.000, C 0.000 }
gfCNCPoint3[13189] = {X 510.9516, Y 64.0089, Z -4.6667, A 0.000, B 0.000, C 0.000 }
gfCNCPoint3[13190] = {X 509.3609, Y 63.0886, Z -4.6667, A 0.000, B 0.000, C 0.000 }
gfCNCPoint3[13191] = {X 507.7389, Y 63.6068, Z -4.6667, A 0.000, B 0.000, C 0.000 }
gfCNCPoint3[13192] = {X 506.0774, Y 63.9798, Z -4.6667, A 0.000, B 0.000, C 0.000 }
gfCNCPoint3[13193] = {X 504.3896, Y 64.2048, Z -4.6667, A 0.000, B 0.000, C 0.000 }
gfCNCPoint3[13194] = {X 502.6885, Y 64.2800, Z -4.6667, A 0.000, B 0.000, C 0.000 }
gfCNCPoint3[13195] = {X 498.4791, Y 64.2800, Z -4.6667, A 0.000, B 0.000, C 0.000 }
gfCNCPoint3[13196] = {X 497.9416, Y 66.2504, Z -4.6667, A 0.000, B 0.000, C 0.000 }
gfCNCPoint3[13197] = {X 497.2391, Y 68.1681, Z -4.6667, A 0.000, B 0.000, C 0.000 }
gfCNCPoint3[13198] = {X 496.3766, Y 70.0195, Z -4.6667, A 0.000, B 0.000, C 0.000 }
gfCNCPoint3[13199] = {X 495.3604, Y 71.7911, Z -4.6667, A 0.000, B 0.000, C 0.000 }
gfCNCPoint3[13200] = {X 495.3605, Y 78.4950, Z -4.6667, A 0.000, B 0.000, C 0.000 }
gfCNCPoint3[13201] = {X 507.6815, Y 78.4950, Z -4.6667, A 0.000, B 0.000, C 0.000 }
gfCNCPoint3[13202] = {X 507.6815, Y 80.8950, Z -4.6667, A 0.000, B 0.000, C 0.000 }
gfCNCPoint3[13203] = {X 580.8966, Y 80.8950, Z -4.6667, A 0.000, B 0.000, C 0.000 }
gfCNCPoint3[13204] = {X 580.8966, Y 68.5934, Z -4.6667, A 0.000, B 0.000, C 0.000 }
gfCNCPoint3[13205] = {X 579.0252, Y 68.4747, Z -4.6667, A 0.000, B 0.000, C 0.000 }
gfCNCPoint3[13206] = {X 577.1691, Y 68.2078, Z -4.6667, A 0.000, B 0.000, C 0.000 }
gfCNCPoint3[13207] = {X 575.3401, Y 67.7943, Z -4.6667, A 0.000, B 0.000, C 0.000 }
gfCNCPoint3[13208] = {X 573.3283, Y 68.2408, Z -4.6667, A 0.000, B 0.000, C 0.000 }
gfCNCPoint3[13209] = {X 571.2852, Y 68.5100, Z -4.6667, A 0.000, B 0.000, C 0.000 }
gfCNCPoint3[13210] = {X 569.2264, Y 68.6000, Z -4.6667, A 0.000, B 0.000, C 0.000 }
gfCNCPoint3[13211] = {X 562.4443, Y 68.6000, Z -4.6667, A 0.000, B 0.000, C 0.000 }
gfCNCPoint3[13212] = {X 560.1443, Y 68.4877, Z -4.6667, A 0.000, B 0.000, C 0.000 }
gfCNCPoint3[13213] = {X 557.8663, Y 68.1517, Z -4.6667, A 0.000, B 0.000, C 0.000 }
gfCNCPoint3[13214] = {X 555.6318, Y 67.5953, Z -4.6667, A 0.000, B 0.000, C 0.000 }
gfCNCPoint3[13215] = {X 553.4621, Y 66.8239, Z -4.6667, A 0.000, B 0.000, C 0.000 }
gfCNCPoint3[13216] = {X 551.3780, Y 65.8446, Z -4.6667, A 0.000, B 0.000, C 0.000 }
gfCNCPoint3[13217] = {X 549.3993, Y 64.6669, Z -4.6667, A 0.000, B 0.000, C 0.000 }
gfCNCPoint3[13218] = {X 547.5447, Y 63.3020, Z -4.6667, A 0.000, B 0.000, C 0.000 }
gfCNCPoint3[13219] = {X 545.8320, Y 61.7628, Z -4.6667, A 0.000, B 0.000, C 0.000 }
gfCNCPoint3[13220] = {X 544.7357, Y 61.8552, Z -4.6667, A 0.000, B 0.000, C 0.000 }
gfCNCPoint3[13221] = {X 543.6358, Y 61.8759, Z -4.6667, A 0.000, B 0.000, C 0.000 }
gfCNCPoint3[13222] = {X 528.1822, Y 61.8763, Z -4.6667, A 0.000, B 0.000, C 0.000 }
gfCNCPoint3[13223] = {X 526.3725, Y 62.6770, Z -4.6667, A 0.000, B 0.000, C 0.000 }
gfCNCPoint3[13224] = {X 524.4820, Y 63.2624, Z -4.6667, A 0.000, B 0.000, C 0.000 }
gfCNCPoint3[13225] = {X 522.5364, Y 63.6247, Z -4.6667, A 0.000, B 0.000, C 0.000 }
gfCNCPoint3[13226] = {X 520.5620, Y 63.7589, Z -4.6667, A 0.000, B 0.000, C 0.000 }
gfCNCPoint3[13227] = {X 519.7998, Y 63.7591, Z -4.6667, A 0.000, B 0.000, C 0.000 }
gfCNCPoint3[13228] = {X 517.9902, Y 63.6618, Z -4.6667, A 0.000, B 0.000, C 0.000 }
gfCNCPoint3[13229] = {X 516.2015, Y 63.3711, Z -4.6667, A 0.000, B 0.000, C 0.000 }
gfCNCPoint3[13230] = {X 514.4543, Y 62.8904, Z -4.6667, A 0.000, B 0.000, C 0.000 }
gfCNCPoint3[13231] = {X 512.7687, Y 62.2251, Z -4.6667, A 0.000, B 0.000, C 0.000 }
gfCNCPoint3[13232] = {X 511.1641, Y 61.3829, Z -4.6667, A 0.000, B 0.000, C 0.000 }
gfCNCPoint3[13233] = {X 509.6590, Y 60.3735, Z -4.6667, A 0.000, B 0.000, C 0.000 }
gfCNCPoint3[13234] = {X 507.9866, Y 61.0270, Z -4.6667, A 0.000, B 0.000, C 0.000 }
gfCNCPoint3[13235] = {X 506.2542, Y 61.4991, Z -4.6667, A 0.000, B 0.000, C 0.000 }
gfCNCPoint3[13236] = {X 504.4815, Y 61.7845, Z -4.6667, A 0.000, B 0.000, C 0.000 }
gfCNCPoint3[13237] = {X 502.6885, Y 61.8800, Z -4.6667, A 0.000, B 0.000, C 0.000 }
gfCNCPoint3[13238] = {X 496.4789, Y 61.8800, Z -4.6667, A 0.000, B 0.000, C 0.000 }
gfCNCPoint3[13239] = {X 496.1192, Y 63.8332, Z -4.6667, A 0.000, B 0.000, C 0.000 }
gfCNCPoint3[13240] = {X 495.5823, Y 65.7453, Z -4.6667, A 0.000, B 0.000, C 0.000 }
gfCNCPoint3[13241] = {X 494.8726, Y 67.6002, Z -4.6667, A 0.000, B 0.000, C 0.000 }
gfCNCPoint3[13242] = {X 493.9962, Y 69.3824, Z -4.6667, A 0.000, B 0.000, C 0.000 }
gfCNCPoint3[13243] = {X 492.9603, Y 71.0769, Z -4.6667, A 0.000, B 0.000, C 0.000 }
gfCNCPoint3[13244] = {X 492.9605, Y 80.8950, Z -4.6667, A 0.000, B 0.000, C 0.000 }
gfCNCPoint3[13245] = {X 507.6815, Y 80.8950, Z -4.6667, A 0.000, B 0.000, C 0.000 }
gfCNCPoint3[13246] = {X 507.6815, Y 83.2950, Z -4.6667, A 0.000, B 0.000, C 0.000 }
gfCNCPoint3[13247] = {X 583.2966, Y 83.2950, Z -4.6667, A 0.000, B 0.000, C 0.000 }
gfCNCPoint3[13248] = {X 583.2966, Y 66.1198, Z -4.6667, A 0.000, B 0.000, C 0.000 }
gfCNCPoint3[13249] = {X 581.2872, Y 66.1993, Z -4.6667, A 0.000, B 0.000, C 0.000 }
gfCNCPoint3[13250] = {X 579.2793, Y 66.0882, Z -4.6667, A 0.000, B 0.000, C 0.000 }
gfCNCPoint3[13251] = {X 577.2910, Y 65.7873, Z -4.6667, A 0.000, B 0.000, C 0.000 }
gfCNCPoint3[13252] = {X 575.3401, Y 65.2993, Z -4.6667, A 0.000, B 0.000, C 0.000 }
gfCNCPoint3[13253] = {X 573.3348, Y 65.7981, Z -4.6667, A 0.000, B 0.000, C 0.000 }
gfCNCPoint3[13254] = {X 571.2904, Y 66.0993, Z -4.6667, A 0.000, B 0.000, C 0.000 }
gfCNCPoint3[13255] = {X 569.2264, Y 66.2000, Z -4.6667, A 0.000, B 0.000, C 0.000 }
gfCNCPoint3[13256] = {X 562.4443, Y 66.2000, Z -4.6667, A 0.000, B 0.000, C 0.000 }
gfCNCPoint3[13257] = {X 560.2303, Y 66.0841, Z -4.6667, A 0.000, B 0.000, C 0.000 }
gfCNCPoint3[13258] = {X 558.0406, Y 65.7376, Z -4.6667, A 0.000, B 0.000, C 0.000 }
gfCNCPoint3[13259] = {X 555.8989, Y 65.1643, Z -4.6667, A 0.000, B 0.000, C 0.000 }
